Fanuc TP program (LS listing): FM195006.ls

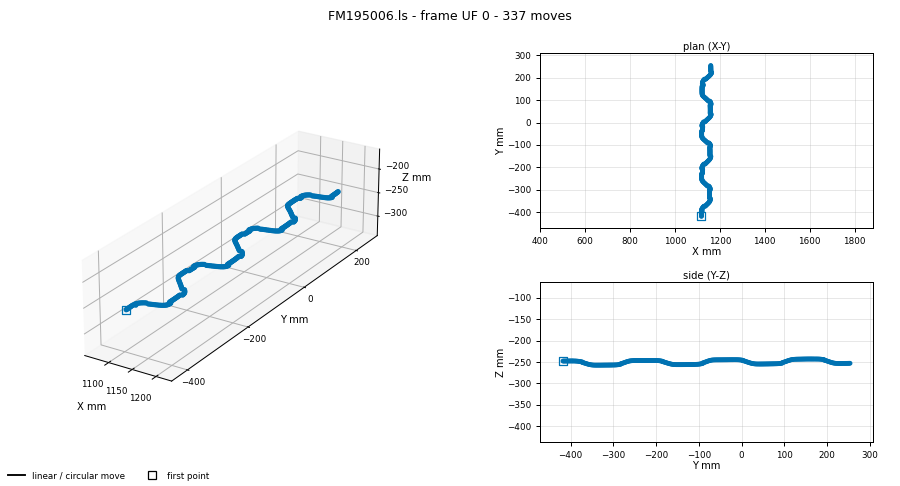
[picture p0: tool path of FM195006.ls in frame UF 0, 337 of 337 moves have a stored position in this frame; points joined in program order, loops and branches not executed]
/PROG  FM195006
/ATTR
OWNER		= MNEDITOR;
COMMENT		= "Auto FANUC move";
PROG_SIZE	= 0;
CREATE		= DATE 26-04-24  TIME 19:50:06;
MODIFIED	= DATE 26-04-24  TIME 19:50:06;
FILE_NAME	= ;
VERSION		= 0;
LINE_COUNT	= 342;
MEMORY_SIZE	= 0;
PROTECT		= READ_WRITE;
TCD:  STACK_SIZE	= 0,
      TASK_PRIORITY	= 50,
      TIME_SLICE	= 0,
      BUSY_LAMP_OFF	= 0,
      ABORT_REQUEST	= 0,
      PAUSE_REQUEST	= 0;
DEFAULT_GROUP	= 1,*,*,*,*;
CONTROL_CODE	= 00000000 00000000;
/MN
   1:  UFRAME_NUM=0 ;
   2:  UTOOL_NUM=1 ;
   3:  R[93]=10 ;
   4:  L P[1] 7mm/sec FINE ;
   5:  L P[2] 7mm/sec FINE ;
   6:  L P[3] 7mm/sec FINE ;
   7:  L P[4] 7mm/sec FINE ;
   8:  L P[5] 7mm/sec FINE ;
   9:  L P[6] 7mm/sec FINE ;
  10:  L P[7] 7mm/sec FINE ;
  11:  L P[8] 7mm/sec FINE ;
  12:  L P[9] 7mm/sec FINE ;
  13:  L P[10] 7mm/sec FINE ;
  14:  L P[11] 7mm/sec FINE ;
  15:  L P[12] 7mm/sec FINE ;
  16:  L P[13] 7mm/sec FINE ;
  17:  L P[14] 7mm/sec FINE ;
  18:  L P[15] 7mm/sec FINE ;
  19:  L P[16] 7mm/sec FINE ;
  20:  L P[17] 7mm/sec FINE ;
  21:  L P[18] 7mm/sec FINE ;
  22:  L P[19] 7mm/sec FINE ;
  23:  L P[20] 7mm/sec FINE ;
  24:  L P[21] 7mm/sec FINE ;
  25:  L P[22] 7mm/sec FINE ;
  26:  L P[23] 7mm/sec FINE ;
  27:  L P[24] 7mm/sec FINE ;
  28:  L P[25] 7mm/sec FINE ;
  29:  L P[26] 7mm/sec FINE ;
  30:  L P[27] 7mm/sec FINE ;
  31:  L P[28] 7mm/sec FINE ;
  32:  L P[29] 7mm/sec FINE ;
  33:  L P[30] 7mm/sec FINE ;
  34:  L P[31] 7mm/sec FINE ;
  35:  L P[32] 7mm/sec FINE ;
  36:  L P[33] 7mm/sec FINE ;
  37:  L P[34] 7mm/sec FINE ;
  38:  L P[35] 7mm/sec FINE ;
  39:  L P[36] 7mm/sec FINE ;
  40:  L P[37] 7mm/sec FINE ;
  41:  L P[38] 7mm/sec FINE ;
  42:  L P[39] 7mm/sec FINE ;
  43:  L P[40] 7mm/sec FINE ;
  44:  L P[41] 7mm/sec FINE ;
  45:  L P[42] 7mm/sec FINE ;
  46:  L P[43] 7mm/sec FINE ;
  47:  L P[44] 7mm/sec FINE ;
  48:  L P[45] 7mm/sec FINE ;
  49:  L P[46] 7mm/sec FINE ;
  50:  L P[47] 7mm/sec FINE ;
  51:  L P[48] 7mm/sec FINE ;
  52:  L P[49] 7mm/sec FINE ;
  53:  L P[50] 7mm/sec FINE ;
  54:  L P[51] 7mm/sec FINE ;
  55:  L P[52] 7mm/sec FINE ;
  56:  L P[53] 7mm/sec FINE ;
  57:  L P[54] 7mm/sec FINE ;
  58:  L P[55] 7mm/sec FINE ;
  59:  L P[56] 7mm/sec FINE ;
  60:  L P[57] 7mm/sec FINE ;
  61:  L P[58] 7mm/sec FINE ;
  62:  L P[59] 7mm/sec FINE ;
  63:  L P[60] 7mm/sec FINE ;
  64:  L P[61] 7mm/sec FINE ;
  65:  L P[62] 7mm/sec FINE ;
  66:  L P[63] 7mm/sec FINE ;
  67:  L P[64] 7mm/sec FINE ;
  68:  L P[65] 7mm/sec FINE ;
  69:  L P[66] 7mm/sec FINE ;
  70:  L P[67] 7mm/sec FINE ;
  71:  L P[68] 7mm/sec FINE ;
  72:  L P[69] 7mm/sec FINE ;
  73:  L P[70] 7mm/sec FINE ;
  74:  L P[71] 7mm/sec FINE ;
  75:  L P[72] 7mm/sec FINE ;
  76:  L P[73] 7mm/sec FINE ;
  77:  L P[74] 7mm/sec FINE ;
  78:  L P[75] 7mm/sec FINE ;
  79:  L P[76] 7mm/sec FINE ;
  80:  L P[77] 7mm/sec FINE ;
  81:  L P[78] 7mm/sec FINE ;
  82:  L P[79] 7mm/sec FINE ;
  83:  L P[80] 7mm/sec FINE ;
  84:  L P[81] 7mm/sec FINE ;
  85:  L P[82] 7mm/sec FINE ;
  86:  L P[83] 7mm/sec FINE ;
  87:  L P[84] 7mm/sec FINE ;
  88:  L P[85] 7mm/sec FINE ;
  89:  L P[86] 7mm/sec FINE ;
  90:  L P[87] 7mm/sec FINE ;
  91:  L P[88] 7mm/sec FINE ;
  92:  L P[89] 7mm/sec FINE ;
  93:  L P[90] 7mm/sec FINE ;
  94:  L P[91] 7mm/sec FINE ;
  95:  L P[92] 7mm/sec FINE ;
  96:  L P[93] 7mm/sec FINE ;
  97:  L P[94] 7mm/sec FINE ;
  98:  L P[95] 7mm/sec FINE ;
  99:  L P[96] 7mm/sec FINE ;
 100:  L P[97] 7mm/sec FINE ;
 101:  L P[98] 7mm/sec FINE ;
 102:  L P[99] 7mm/sec FINE ;
 103:  L P[100] 7mm/sec FINE ;
 104:  L P[101] 7mm/sec FINE ;
 105:  L P[102] 7mm/sec FINE ;
 106:  L P[103] 7mm/sec FINE ;
 107:  L P[104] 7mm/sec FINE ;
 108:  L P[105] 7mm/sec FINE ;
 109:  L P[106] 7mm/sec FINE ;
 110:  L P[107] 7mm/sec FINE ;
 111:  L P[108] 7mm/sec FINE ;
 112:  L P[109] 7mm/sec FINE ;
 113:  L P[110] 7mm/sec FINE ;
 114:  L P[111] 7mm/sec FINE ;
 115:  L P[112] 7mm/sec FINE ;
 116:  L P[113] 7mm/sec FINE ;
 117:  L P[114] 7mm/sec FINE ;
 118:  L P[115] 7mm/sec FINE ;
 119:  L P[116] 7mm/sec FINE ;
 120:  L P[117] 7mm/sec FINE ;
 121:  L P[118] 7mm/sec FINE ;
 122:  L P[119] 7mm/sec FINE ;
 123:  L P[120] 7mm/sec FINE ;
 124:  L P[121] 7mm/sec FINE ;
 125:  L P[122] 7mm/sec FINE ;
 126:  L P[123] 7mm/sec FINE ;
 127:  L P[124] 7mm/sec FINE ;
 128:  L P[125] 7mm/sec FINE ;
 129:  L P[126] 7mm/sec FINE ;
 130:  L P[127] 7mm/sec FINE ;
 131:  L P[128] 7mm/sec FINE ;
 132:  L P[129] 7mm/sec FINE ;
 133:  L P[130] 7mm/sec FINE ;
 134:  L P[131] 7mm/sec FINE ;
 135:  L P[132] 7mm/sec FINE ;
 136:  L P[133] 7mm/sec FINE ;
 137:  L P[134] 7mm/sec FINE ;
 138:  L P[135] 7mm/sec FINE ;
 139:  L P[136] 7mm/sec FINE ;
 140:  L P[137] 7mm/sec FINE ;
 141:  L P[138] 7mm/sec FINE ;
 142:  L P[139] 7mm/sec FINE ;
 143:  L P[140] 7mm/sec FINE ;
 144:  L P[141] 7mm/sec FINE ;
 145:  L P[142] 7mm/sec FINE ;
 146:  L P[143] 7mm/sec FINE ;
 147:  L P[144] 7mm/sec FINE ;
 148:  L P[145] 7mm/sec FINE ;
 149:  L P[146] 7mm/sec FINE ;
 150:  L P[147] 7mm/sec FINE ;
 151:  L P[148] 7mm/sec FINE ;
 152:  L P[149] 7mm/sec FINE ;
 153:  L P[150] 7mm/sec FINE ;
 154:  L P[151] 7mm/sec FINE ;
 155:  L P[152] 7mm/sec FINE ;
 156:  L P[153] 7mm/sec FINE ;
 157:  L P[154] 7mm/sec FINE ;
 158:  L P[155] 7mm/sec FINE ;
 159:  L P[156] 7mm/sec FINE ;
 160:  L P[157] 7mm/sec FINE ;
 161:  L P[158] 7mm/sec FINE ;
 162:  L P[159] 7mm/sec FINE ;
 163:  L P[160] 7mm/sec FINE ;
 164:  L P[161] 7mm/sec FINE ;
 165:  L P[162] 7mm/sec FINE ;
 166:  L P[163] 7mm/sec FINE ;
 167:  L P[164] 7mm/sec FINE ;
 168:  L P[165] 7mm/sec FINE ;
 169:  L P[166] 7mm/sec FINE ;
 170:  L P[167] 7mm/sec FINE ;
 171:  L P[168] 7mm/sec FINE ;
 172:  L P[169] 7mm/sec FINE ;
 173:  L P[170] 7mm/sec FINE ;
 174:  L P[171] 7mm/sec FINE ;
 175:  L P[172] 7mm/sec FINE ;
 176:  L P[173] 7mm/sec FINE ;
 177:  L P[174] 7mm/sec FINE ;
 178:  L P[175] 7mm/sec FINE ;
 179:  L P[176] 7mm/sec FINE ;
 180:  L P[177] 7mm/sec FINE ;
 181:  L P[178] 7mm/sec FINE ;
 182:  L P[179] 7mm/sec FINE ;
 183:  L P[180] 7mm/sec FINE ;
 184:  L P[181] 7mm/sec FINE ;
 185:  L P[182] 7mm/sec FINE ;
 186:  L P[183] 7mm/sec FINE ;
 187:  L P[184] 7mm/sec FINE ;
 188:  L P[185] 7mm/sec FINE ;
 189:  L P[186] 7mm/sec FINE ;
 190:  L P[187] 7mm/sec FINE ;
 191:  L P[188] 7mm/sec FINE ;
 192:  L P[189] 7mm/sec FINE ;
 193:  L P[190] 7mm/sec FINE ;
 194:  L P[191] 7mm/sec FINE ;
 195:  L P[192] 7mm/sec FINE ;
 196:  L P[193] 7mm/sec FINE ;
 197:  L P[194] 7mm/sec FINE ;
 198:  L P[195] 7mm/sec FINE ;
 199:  L P[196] 7mm/sec FINE ;
 200:  L P[197] 7mm/sec FINE ;
 201:  L P[198] 7mm/sec FINE ;
 202:  L P[199] 7mm/sec FINE ;
 203:  L P[200] 7mm/sec FINE ;
 204:  L P[201] 7mm/sec FINE ;
 205:  L P[202] 7mm/sec FINE ;
 206:  L P[203] 7mm/sec FINE ;
 207:  L P[204] 7mm/sec FINE ;
 208:  L P[205] 7mm/sec FINE ;
 209:  L P[206] 7mm/sec FINE ;
 210:  L P[207] 7mm/sec FINE ;
 211:  L P[208] 7mm/sec FINE ;
 212:  L P[209] 7mm/sec FINE ;
 213:  L P[210] 7mm/sec FINE ;
 214:  L P[211] 7mm/sec FINE ;
 215:  L P[212] 7mm/sec FINE ;
 216:  L P[213] 7mm/sec FINE ;
 217:  L P[214] 7mm/sec FINE ;
 218:  L P[215] 7mm/sec FINE ;
 219:  L P[216] 7mm/sec FINE ;
 220:  L P[217] 7mm/sec FINE ;
 221:  L P[218] 7mm/sec FINE ;
 222:  L P[219] 7mm/sec FINE ;
 223:  L P[220] 7mm/sec FINE ;
 224:  L P[221] 7mm/sec FINE ;
 225:  L P[222] 7mm/sec FINE ;
 226:  L P[223] 7mm/sec FINE ;
 227:  L P[224] 7mm/sec FINE ;
 228:  L P[225] 7mm/sec FINE ;
 229:  L P[226] 7mm/sec FINE ;
 230:  L P[227] 7mm/sec FINE ;
 231:  L P[228] 7mm/sec FINE ;
 232:  L P[229] 7mm/sec FINE ;
 233:  L P[230] 7mm/sec FINE ;
 234:  L P[231] 7mm/sec FINE ;
 235:  L P[232] 7mm/sec FINE ;
 236:  L P[233] 7mm/sec FINE ;
 237:  L P[234] 7mm/sec FINE ;
 238:  L P[235] 7mm/sec FINE ;
 239:  L P[236] 7mm/sec FINE ;
 240:  L P[237] 7mm/sec FINE ;
 241:  L P[238] 7mm/sec FINE ;
 242:  L P[239] 7mm/sec FINE ;
 243:  L P[240] 7mm/sec FINE ;
 244:  L P[241] 7mm/sec FINE ;
 245:  L P[242] 7mm/sec FINE ;
 246:  L P[243] 7mm/sec FINE ;
 247:  L P[244] 7mm/sec FINE ;
 248:  L P[245] 7mm/sec FINE ;
 249:  L P[246] 7mm/sec FINE ;
 250:  L P[247] 7mm/sec FINE ;
 251:  L P[248] 7mm/sec FINE ;
 252:  L P[249] 7mm/sec FINE ;
 253:  L P[250] 7mm/sec FINE ;
 254:  L P[251] 7mm/sec FINE ;
 255:  L P[252] 7mm/sec FINE ;
 256:  L P[253] 7mm/sec FINE ;
 257:  L P[254] 7mm/sec FINE ;
 258:  L P[255] 7mm/sec FINE ;
 259:  L P[256] 7mm/sec FINE ;
 260:  L P[257] 7mm/sec FINE ;
 261:  L P[258] 7mm/sec FINE ;
 262:  L P[259] 7mm/sec FINE ;
 263:  L P[260] 7mm/sec FINE ;
 264:  L P[261] 7mm/sec FINE ;
 265:  L P[262] 7mm/sec FINE ;
 266:  L P[263] 7mm/sec FINE ;
 267:  L P[264] 7mm/sec FINE ;
 268:  L P[265] 7mm/sec FINE ;
 269:  L P[266] 7mm/sec FINE ;
 270:  L P[267] 7mm/sec FINE ;
 271:  L P[268] 7mm/sec FINE ;
 272:  L P[269] 7mm/sec FINE ;
 273:  L P[270] 7mm/sec FINE ;
 274:  L P[271] 7mm/sec FINE ;
 275:  L P[272] 7mm/sec FINE ;
 276:  L P[273] 7mm/sec FINE ;
 277:  L P[274] 7mm/sec FINE ;
 278:  L P[275] 7mm/sec FINE ;
 279:  L P[276] 7mm/sec FINE ;
 280:  L P[277] 7mm/sec FINE ;
 281:  L P[278] 7mm/sec FINE ;
 282:  L P[279] 7mm/sec FINE ;
 283:  L P[280] 7mm/sec FINE ;
 284:  L P[281] 7mm/sec FINE ;
 285:  L P[282] 7mm/sec FINE ;
 286:  L P[283] 7mm/sec FINE ;
 287:  L P[284] 7mm/sec FINE ;
 288:  L P[285] 7mm/sec FINE ;
 289:  L P[286] 7mm/sec FINE ;
 290:  L P[287] 7mm/sec FINE ;
 291:  L P[288] 7mm/sec FINE ;
 292:  L P[289] 7mm/sec FINE ;
 293:  L P[290] 7mm/sec FINE ;
 294:  L P[291] 7mm/sec FINE ;
 295:  L P[292] 7mm/sec FINE ;
 296:  L P[293] 7mm/sec FINE ;
 297:  L P[294] 7mm/sec FINE ;
 298:  L P[295] 7mm/sec FINE ;
 299:  L P[296] 7mm/sec FINE ;
 300:  L P[297] 7mm/sec FINE ;
 301:  L P[298] 7mm/sec FINE ;
 302:  L P[299] 7mm/sec FINE ;
 303:  L P[300] 7mm/sec FINE ;
 304:  L P[301] 7mm/sec FINE ;
 305:  L P[302] 7mm/sec FINE ;
 306:  L P[303] 7mm/sec FINE ;
 307:  L P[304] 7mm/sec FINE ;
 308:  L P[305] 7mm/sec FINE ;
 309:  L P[306] 7mm/sec FINE ;
 310:  L P[307] 7mm/sec FINE ;
 311:  L P[308] 7mm/sec FINE ;
 312:  L P[309] 7mm/sec FINE ;
 313:  L P[310] 7mm/sec FINE ;
 314:  L P[311] 7mm/sec FINE ;
 315:  L P[312] 7mm/sec FINE ;
 316:  L P[313] 7mm/sec FINE ;
 317:  L P[314] 7mm/sec FINE ;
 318:  L P[315] 7mm/sec FINE ;
 319:  L P[316] 7mm/sec FINE ;
 320:  L P[317] 7mm/sec FINE ;
 321:  L P[318] 7mm/sec FINE ;
 322:  L P[319] 7mm/sec FINE ;
 323:  L P[320] 7mm/sec FINE ;
 324:  L P[321] 7mm/sec FINE ;
 325:  L P[322] 7mm/sec FINE ;
 326:  L P[323] 7mm/sec FINE ;
 327:  L P[324] 7mm/sec FINE ;
 328:  L P[325] 7mm/sec FINE ;
 329:  L P[326] 7mm/sec FINE ;
 330:  L P[327] 7mm/sec FINE ;
 331:  L P[328] 7mm/sec FINE ;
 332:  L P[329] 7mm/sec FINE ;
 333:  L P[330] 7mm/sec FINE ;
 334:  L P[331] 7mm/sec FINE ;
 335:  L P[332] 7mm/sec FINE ;
 336:  L P[333] 7mm/sec FINE ;
 337:  L P[334] 7mm/sec FINE ;
 338:  L P[335] 7mm/sec FINE ;
 339:  L P[336] 7mm/sec FINE ;
 340:  L P[337] 7mm/sec FINE ;
 341:  R[93]=1 ;
 342:  END ;
/POS
P[1]{
   GP1:
	UF : 0, UT : 1,		CONFIG : 'N U T, 0, 0, 0',
	X = 1117.999  mm,	Y = -418.067  mm,	Z = -247.754  mm,
	W = 0.000 deg,	P = 30.000 deg,	R = 175.494 deg
};
P[2]{
   GP1:
	UF : 0, UT : 1,		CONFIG : 'N U T, 0, 0, 0',
	X = 1117.932  mm,	Y = -416.071  mm,	Z = -247.733  mm,
	W = 0.000 deg,	P = 30.000 deg,	R = 175.494 deg
};
P[3]{
   GP1:
	UF : 0, UT : 1,		CONFIG : 'N U T, 0, 0, 0',
	X = 1117.857  mm,	Y = -414.076  mm,	Z = -247.707  mm,
	W = 0.000 deg,	P = 30.000 deg,	R = 175.494 deg
};
P[4]{
   GP1:
	UF : 0, UT : 1,		CONFIG : 'N U T, 0, 0, 0',
	X = 1117.780  mm,	Y = -412.071  mm,	Z = -247.675  mm,
	W = 0.000 deg,	P = 30.000 deg,	R = 175.494 deg
};
P[5]{
   GP1:
	UF : 0, UT : 1,		CONFIG : 'N U T, 0, 0, 0',
	X = 1117.714  mm,	Y = -410.060  mm,	Z = -247.642  mm,
	W = 0.000 deg,	P = 30.000 deg,	R = 175.494 deg
};
P[6]{
   GP1:
	UF : 0, UT : 1,		CONFIG : 'N U T, 0, 0, 0',
	X = 1117.659  mm,	Y = -408.049  mm,	Z = -247.610  mm,
	W = 0.000 deg,	P = 30.000 deg,	R = 175.494 deg
};
P[7]{
   GP1:
	UF : 0, UT : 1,		CONFIG : 'N U T, 0, 0, 0',
	X = 1117.615  mm,	Y = -406.039  mm,	Z = -247.582  mm,
	W = 0.000 deg,	P = 30.000 deg,	R = 175.494 deg
};
P[8]{
   GP1:
	UF : 0, UT : 1,		CONFIG : 'N U T, 0, 0, 0',
	X = 1117.582  mm,	Y = -404.022  mm,	Z = -247.555  mm,
	W = 0.000 deg,	P = 30.000 deg,	R = 175.494 deg
};
P[9]{
   GP1:
	UF : 0, UT : 1,		CONFIG : 'N U T, 0, 0, 0',
	X = 1117.571  mm,	Y = -402.004  mm,	Z = -247.531  mm,
	W = 0.000 deg,	P = 30.000 deg,	R = 175.494 deg
};
P[10]{
   GP1:
	UF : 0, UT : 1,		CONFIG : 'N U T, 0, 0, 0',
	X = 1117.574  mm,	Y = -399.980  mm,	Z = -247.513  mm,
	W = 0.000 deg,	P = 30.000 deg,	R = 175.494 deg
};
P[11]{
   GP1:
	UF : 0, UT : 1,		CONFIG : 'N U T, 0, 0, 0',
	X = 1117.612  mm,	Y = -397.943  mm,	Z = -247.507  mm,
	W = 0.000 deg,	P = 30.000 deg,	R = 175.494 deg
};
P[12]{
   GP1:
	UF : 0, UT : 1,		CONFIG : 'N U T, 0, 0, 0',
	X = 1117.692  mm,	Y = -395.874  mm,	Z = -247.515  mm,
	W = 0.000 deg,	P = 30.000 deg,	R = 175.494 deg
};
P[13]{
   GP1:
	UF : 0, UT : 1,		CONFIG : 'N U T, 0, 0, 0',
	X = 1121.852  mm,	Y = -394.217  mm,	Z = -247.538  mm,
	W = 0.000 deg,	P = 30.000 deg,	R = 175.494 deg
};
P[14]{
   GP1:
	UF : 0, UT : 1,		CONFIG : 'N U T, 0, 0, 0',
	X = 1118.152  mm,	Y = -391.671  mm,	Z = -247.590  mm,
	W = 0.000 deg,	P = 30.000 deg,	R = 170.031 deg
};
P[15]{
   GP1:
	UF : 0, UT : 1,		CONFIG : 'N U T, 0, 0, 0',
	X = 1118.595  mm,	Y = -389.498  mm,	Z = -247.675  mm,
	W = 0.000 deg,	P = 30.000 deg,	R = 162.233 deg
};
P[16]{
   GP1:
	UF : 0, UT : 1,		CONFIG : 'N U T, 0, 0, 0',
	X = 1119.280  mm,	Y = -387.326  mm,	Z = -247.802  mm,
	W = 0.000 deg,	P = 30.000 deg,	R = 154.209 deg
};
P[17]{
   GP1:
	UF : 0, UT : 1,		CONFIG : 'N U T, 0, 0, 0',
	X = 1120.146  mm,	Y = -385.162  mm,	Z = -247.954  mm,
	W = 0.000 deg,	P = 30.000 deg,	R = 145.966 deg
};
P[18]{
   GP1:
	UF : 0, UT : 1,		CONFIG : 'N U T, 0, 0, 0',
	X = 1121.277  mm,	Y = -383.000  mm,	Z = -248.156  mm,
	W = 0.000 deg,	P = 30.000 deg,	R = 137.314 deg
};
P[19]{
   GP1:
	UF : 0, UT : 1,		CONFIG : 'N U T, 0, 0, 0',
	X = 1122.601  mm,	Y = -380.901  mm,	Z = -248.418  mm,
	W = 0.000 deg,	P = 30.000 deg,	R = 137.314 deg
};
P[20]{
   GP1:
	UF : 0, UT : 1,		CONFIG : 'N U T, 0, 0, 0',
	X = 1124.026  mm,	Y = -378.816  mm,	Z = -248.729  mm,
	W = 0.000 deg,	P = 30.000 deg,	R = 137.314 deg
};
P[21]{
   GP1:
	UF : 0, UT : 1,		CONFIG : 'N U T, 0, 0, 0',
	X = 1125.669  mm,	Y = -376.727  mm,	Z = -249.118  mm,
	W = 0.000 deg,	P = 30.000 deg,	R = 137.314 deg
};
P[22]{
   GP1:
	UF : 0, UT : 1,		CONFIG : 'N U T, 0, 0, 0',
	X = 1127.425  mm,	Y = -374.692  mm,	Z = -249.568  mm,
	W = 0.000 deg,	P = 30.000 deg,	R = 137.314 deg
};
P[23]{
   GP1:
	UF : 0, UT : 1,		CONFIG : 'N U T, 0, 0, 0',
	X = 1129.189  mm,	Y = -372.655  mm,	Z = -250.051  mm,
	W = 0.000 deg,	P = 30.000 deg,	R = 137.314 deg
};
P[24]{
   GP1:
	UF : 0, UT : 1,		CONFIG : 'N U T, 0, 0, 0',
	X = 1134.014  mm,	Y = -373.387  mm,	Z = -250.615  mm,
	W = 0.000 deg,	P = 30.000 deg,	R = 137.314 deg
};
P[25]{
   GP1:
	UF : 0, UT : 1,		CONFIG : 'N U T, 0, 0, 0',
	X = 1135.950  mm,	Y = -371.401  mm,	Z = -251.227  mm,
	W = 0.000 deg,	P = 30.000 deg,	R = 137.314 deg
};
P[26]{
   GP1:
	UF : 0, UT : 1,		CONFIG : 'N U T, 0, 0, 0',
	X = 1137.893  mm,	Y = -369.434  mm,	Z = -251.859  mm,
	W = 0.000 deg,	P = 30.000 deg,	R = 137.314 deg
};
P[27]{
   GP1:
	UF : 0, UT : 1,		CONFIG : 'N U T, 0, 0, 0',
	X = 1140.018  mm,	Y = -367.445  mm,	Z = -252.527  mm,
	W = 0.000 deg,	P = 30.000 deg,	R = 137.314 deg
};
P[28]{
   GP1:
	UF : 0, UT : 1,		CONFIG : 'N U T, 0, 0, 0',
	X = 1142.083  mm,	Y = -365.426  mm,	Z = -253.157  mm,
	W = 0.000 deg,	P = 30.000 deg,	R = 137.314 deg
};
P[29]{
   GP1:
	UF : 0, UT : 1,		CONFIG : 'N U T, 0, 0, 0',
	X = 1144.092  mm,	Y = -363.439  mm,	Z = -253.772  mm,
	W = 0.000 deg,	P = 30.000 deg,	R = 137.314 deg
};
P[30]{
   GP1:
	UF : 0, UT : 1,		CONFIG : 'N U T, 0, 0, 0',
	X = 1146.210  mm,	Y = -361.441  mm,	Z = -254.406  mm,
	W = 0.000 deg,	P = 30.000 deg,	R = 143.831 deg
};
P[31]{
   GP1:
	UF : 0, UT : 1,		CONFIG : 'N U T, 0, 0, 0',
	X = 1148.286  mm,	Y = -359.401  mm,	Z = -255.004  mm,
	W = 0.000 deg,	P = 30.000 deg,	R = 155.941 deg
};
P[32]{
   GP1:
	UF : 0, UT : 1,		CONFIG : 'N U T, 0, 0, 0',
	X = 1150.228  mm,	Y = -357.348  mm,	Z = -255.551  mm,
	W = 0.000 deg,	P = 30.000 deg,	R = 167.597 deg
};
P[33]{
   GP1:
	UF : 0, UT : 1,		CONFIG : 'N U T, 0, 0, 0',
	X = 1152.071  mm,	Y = -355.248  mm,	Z = -256.048  mm,
	W = 0.000 deg,	P = 30.000 deg,	R = 178.845 deg
};
P[34]{
   GP1:
	UF : 0, UT : 1,		CONFIG : 'N U T, 0, 0, 0',
	X = 1153.605  mm,	Y = -353.112  mm,	Z = -256.446  mm,
	W = 0.000 deg,	P = 30.000 deg,	R = 178.845 deg
};
P[35]{
   GP1:
	UF : 0, UT : 1,		CONFIG : 'N U T, 0, 0, 0',
	X = 1154.932  mm,	Y = -350.971  mm,	Z = -256.780  mm,
	W = 0.000 deg,	P = 30.000 deg,	R = 178.845 deg
};
P[36]{
   GP1:
	UF : 0, UT : 1,		CONFIG : 'N U T, 0, 0, 0',
	X = 1156.016  mm,	Y = -348.756  mm,	Z = -257.035  mm,
	W = 0.000 deg,	P = 30.000 deg,	R = 178.845 deg
};
P[37]{
   GP1:
	UF : 0, UT : 1,		CONFIG : 'N U T, 0, 0, 0',
	X = 1156.751  mm,	Y = -346.509  mm,	Z = -257.195  mm,
	W = 0.000 deg,	P = 30.000 deg,	R = 178.845 deg
};
P[38]{
   GP1:
	UF : 0, UT : 1,		CONFIG : 'N U T, 0, 0, 0',
	X = 1157.193  mm,	Y = -344.312  mm,	Z = -257.285  mm,
	W = 0.000 deg,	P = 30.000 deg,	R = 178.845 deg
};
P[39]{
   GP1:
	UF : 0, UT : 1,		CONFIG : 'N U T, 0, 0, 0',
	X = 1157.443  mm,	Y = -342.157  mm,	Z = -257.325  mm,
	W = 0.000 deg,	P = 30.000 deg,	R = 178.845 deg
};
P[40]{
   GP1:
	UF : 0, UT : 1,		CONFIG : 'N U T, 0, 0, 0',
	X = 1157.532  mm,	Y = -340.068  mm,	Z = -257.329  mm,
	W = 0.000 deg,	P = 30.000 deg,	R = 178.845 deg
};
P[41]{
   GP1:
	UF : 0, UT : 1,		CONFIG : 'N U T, 0, 0, 0',
	X = 1157.585  mm,	Y = -338.048  mm,	Z = -257.329  mm,
	W = 0.000 deg,	P = 30.000 deg,	R = 178.845 deg
};
P[42]{
   GP1:
	UF : 0, UT : 1,		CONFIG : 'N U T, 0, 0, 0',
	X = 1153.629  mm,	Y = -335.963  mm,	Z = -257.326  mm,
	W = 0.000 deg,	P = 30.000 deg,	R = 178.845 deg
};
P[43]{
   GP1:
	UF : 0, UT : 1,		CONFIG : 'N U T, 0, 0, 0',
	X = 1153.660  mm,	Y = -333.972  mm,	Z = -257.321  mm,
	W = 0.000 deg,	P = 30.000 deg,	R = 178.845 deg
};
P[44]{
   GP1:
	UF : 0, UT : 1,		CONFIG : 'N U T, 0, 0, 0',
	X = 1153.684  mm,	Y = -331.978  mm,	Z = -257.311  mm,
	W = 0.000 deg,	P = 30.000 deg,	R = 178.845 deg
};
P[45]{
   GP1:
	UF : 0, UT : 1,		CONFIG : 'N U T, 0, 0, 0',
	X = 1153.703  mm,	Y = -329.986  mm,	Z = -257.295  mm,
	W = 0.000 deg,	P = 30.000 deg,	R = 178.845 deg
};
P[46]{
   GP1:
	UF : 0, UT : 1,		CONFIG : 'N U T, 0, 0, 0',
	X = 1153.712  mm,	Y = -327.993  mm,	Z = -257.277  mm,
	W = 0.000 deg,	P = 30.000 deg,	R = 178.845 deg
};
P[47]{
   GP1:
	UF : 0, UT : 1,		CONFIG : 'N U T, 0, 0, 0',
	X = 1153.716  mm,	Y = -325.996  mm,	Z = -257.255  mm,
	W = 0.000 deg,	P = 30.000 deg,	R = 178.845 deg
};
P[48]{
   GP1:
	UF : 0, UT : 1,		CONFIG : 'N U T, 0, 0, 0',
	X = 1153.719  mm,	Y = -323.998  mm,	Z = -257.232  mm,
	W = 0.000 deg,	P = 30.000 deg,	R = 178.845 deg
};
P[49]{
   GP1:
	UF : 0, UT : 1,		CONFIG : 'N U T, 0, 0, 0',
	X = 1153.721  mm,	Y = -321.999  mm,	Z = -257.210  mm,
	W = 0.000 deg,	P = 30.000 deg,	R = 178.845 deg
};
P[50]{
   GP1:
	UF : 0, UT : 1,		CONFIG : 'N U T, 0, 0, 0',
	X = 1153.721  mm,	Y = -320.005  mm,	Z = -257.188  mm,
	W = 0.000 deg,	P = 30.000 deg,	R = 178.845 deg
};
P[51]{
   GP1:
	UF : 0, UT : 1,		CONFIG : 'N U T, 0, 0, 0',
	X = 1153.710  mm,	Y = -318.013  mm,	Z = -257.169  mm,
	W = 0.000 deg,	P = 30.000 deg,	R = 178.845 deg
};
P[52]{
   GP1:
	UF : 0, UT : 1,		CONFIG : 'N U T, 0, 0, 0',
	X = 1153.695  mm,	Y = -316.020  mm,	Z = -257.154  mm,
	W = 0.000 deg,	P = 30.000 deg,	R = 178.845 deg
};
P[53]{
   GP1:
	UF : 0, UT : 1,		CONFIG : 'N U T, 0, 0, 0',
	X = 1153.671  mm,	Y = -314.026  mm,	Z = -257.140  mm,
	W = 0.000 deg,	P = 30.000 deg,	R = 178.845 deg
};
P[54]{
   GP1:
	UF : 0, UT : 1,		CONFIG : 'N U T, 0, 0, 0',
	X = 1153.644  mm,	Y = -312.033  mm,	Z = -257.124  mm,
	W = 0.000 deg,	P = 30.000 deg,	R = 178.845 deg
};
P[55]{
   GP1:
	UF : 0, UT : 1,		CONFIG : 'N U T, 0, 0, 0',
	X = 1153.605  mm,	Y = -310.048  mm,	Z = -257.107  mm,
	W = 0.000 deg,	P = 30.000 deg,	R = 178.845 deg
};
P[56]{
   GP1:
	UF : 0, UT : 1,		CONFIG : 'N U T, 0, 0, 0',
	X = 1153.548  mm,	Y = -308.060  mm,	Z = -257.086  mm,
	W = 0.000 deg,	P = 30.000 deg,	R = 178.845 deg
};
P[57]{
   GP1:
	UF : 0, UT : 1,		CONFIG : 'N U T, 0, 0, 0',
	X = 1153.485  mm,	Y = -306.064  mm,	Z = -257.062  mm,
	W = 0.000 deg,	P = 30.000 deg,	R = 178.845 deg
};
P[58]{
   GP1:
	UF : 0, UT : 1,		CONFIG : 'N U T, 0, 0, 0',
	X = 1153.421  mm,	Y = -304.072  mm,	Z = -257.034  mm,
	W = 0.000 deg,	P = 30.000 deg,	R = 178.845 deg
};
P[59]{
   GP1:
	UF : 0, UT : 1,		CONFIG : 'N U T, 0, 0, 0',
	X = 1153.342  mm,	Y = -302.082  mm,	Z = -257.003  mm,
	W = 0.000 deg,	P = 30.000 deg,	R = 178.845 deg
};
P[60]{
   GP1:
	UF : 0, UT : 1,		CONFIG : 'N U T, 0, 0, 0',
	X = 1157.251  mm,	Y = -299.879  mm,	Z = -256.967  mm,
	W = 0.000 deg,	P = 30.000 deg,	R = -172.841 deg
};
P[61]{
   GP1:
	UF : 0, UT : 1,		CONFIG : 'N U T, 0, 0, 0',
	X = 1157.091  mm,	Y = -297.823  mm,	Z = -256.913  mm,
	W = 0.000 deg,	P = 30.000 deg,	R = -163.968 deg
};
P[62]{
   GP1:
	UF : 0, UT : 1,		CONFIG : 'N U T, 0, 0, 0',
	X = 1156.883  mm,	Y = -295.745  mm,	Z = -256.846  mm,
	W = 0.000 deg,	P = 30.000 deg,	R = -155.076 deg
};
P[63]{
   GP1:
	UF : 0, UT : 1,		CONFIG : 'N U T, 0, 0, 0',
	X = 1156.543  mm,	Y = -293.588  mm,	Z = -256.745  mm,
	W = 0.000 deg,	P = 30.000 deg,	R = -146.113 deg
};
P[64]{
   GP1:
	UF : 0, UT : 1,		CONFIG : 'N U T, 0, 0, 0',
	X = 1155.946  mm,	Y = -291.342  mm,	Z = -256.580  mm,
	W = 0.000 deg,	P = 30.000 deg,	R = -136.938 deg
};
P[65]{
   GP1:
	UF : 0, UT : 1,		CONFIG : 'N U T, 0, 0, 0',
	X = 1154.950  mm,	Y = -289.046  mm,	Z = -256.318  mm,
	W = 0.000 deg,	P = 30.000 deg,	R = -136.938 deg
};
P[66]{
   GP1:
	UF : 0, UT : 1,		CONFIG : 'N U T, 0, 0, 0',
	X = 1153.530  mm,	Y = -286.860  mm,	Z = -255.916  mm,
	W = 0.000 deg,	P = 30.000 deg,	R = -136.938 deg
};
P[67]{
   GP1:
	UF : 0, UT : 1,		CONFIG : 'N U T, 0, 0, 0',
	X = 1151.985  mm,	Y = -284.759  mm,	Z = -255.467  mm,
	W = 0.000 deg,	P = 30.000 deg,	R = -136.938 deg
};
P[68]{
   GP1:
	UF : 0, UT : 1,		CONFIG : 'N U T, 0, 0, 0',
	X = 1150.225  mm,	Y = -282.682  mm,	Z = -254.945  mm,
	W = 0.000 deg,	P = 30.000 deg,	R = -136.938 deg
};
P[69]{
   GP1:
	UF : 0, UT : 1,		CONFIG : 'N U T, 0, 0, 0',
	X = 1145.453  mm,	Y = -283.369  mm,	Z = -254.386  mm,
	W = 0.000 deg,	P = 30.000 deg,	R = -136.938 deg
};
P[70]{
   GP1:
	UF : 0, UT : 1,		CONFIG : 'N U T, 0, 0, 0',
	X = 1143.577  mm,	Y = -281.438  mm,	Z = -253.781  mm,
	W = 0.000 deg,	P = 30.000 deg,	R = -136.938 deg
};
P[71]{
   GP1:
	UF : 0, UT : 1,		CONFIG : 'N U T, 0, 0, 0',
	X = 1141.392  mm,	Y = -279.447  mm,	Z = -253.092  mm,
	W = 0.000 deg,	P = 30.000 deg,	R = -136.938 deg
};
P[72]{
   GP1:
	UF : 0, UT : 1,		CONFIG : 'N U T, 0, 0, 0',
	X = 1139.366  mm,	Y = -277.421  mm,	Z = -252.452  mm,
	W = 0.000 deg,	P = 30.000 deg,	R = -136.938 deg
};
P[73]{
   GP1:
	UF : 0, UT : 1,		CONFIG : 'N U T, 0, 0, 0',
	X = 1137.351  mm,	Y = -275.446  mm,	Z = -251.780  mm,
	W = 0.000 deg,	P = 30.000 deg,	R = -136.938 deg
};
P[74]{
   GP1:
	UF : 0, UT : 1,		CONFIG : 'N U T, 0, 0, 0',
	X = 1135.216  mm,	Y = -273.455  mm,	Z = -251.043  mm,
	W = 0.000 deg,	P = 30.000 deg,	R = -136.938 deg
};
P[75]{
   GP1:
	UF : 0, UT : 1,		CONFIG : 'N U T, 0, 0, 0',
	X = 1133.147  mm,	Y = -271.482  mm,	Z = -250.323  mm,
	W = 0.000 deg,	P = 30.000 deg,	R = -136.938 deg
};
P[76]{
   GP1:
	UF : 0, UT : 1,		CONFIG : 'N U T, 0, 0, 0',
	X = 1130.846  mm,	Y = -269.496  mm,	Z = -249.596  mm,
	W = 0.000 deg,	P = 30.000 deg,	R = -136.938 deg
};
P[77]{
   GP1:
	UF : 0, UT : 1,		CONFIG : 'N U T, 0, 0, 0',
	X = 1128.600  mm,	Y = -267.443  mm,	Z = -248.935  mm,
	W = 0.000 deg,	P = 30.000 deg,	R = -144.465 deg
};
P[78]{
   GP1:
	UF : 0, UT : 1,		CONFIG : 'N U T, 0, 0, 0',
	X = 1126.581  mm,	Y = -265.403  mm,	Z = -248.356  mm,
	W = 0.000 deg,	P = 30.000 deg,	R = -156.971 deg
};
P[79]{
   GP1:
	UF : 0, UT : 1,		CONFIG : 'N U T, 0, 0, 0',
	X = 1124.538  mm,	Y = -263.312  mm,	Z = -247.787  mm,
	W = 0.000 deg,	P = 30.000 deg,	R = -169.411 deg
};
P[80]{
   GP1:
	UF : 0, UT : 1,		CONFIG : 'N U T, 0, 0, 0',
	X = 1122.883  mm,	Y = -261.136  mm,	Z = -247.389  mm,
	W = 0.000 deg,	P = 30.000 deg,	R = 179.517 deg
};
P[81]{
   GP1:
	UF : 0, UT : 1,		CONFIG : 'N U T, 0, 0, 0',
	X = 1121.541  mm,	Y = -258.975  mm,	Z = -247.111  mm,
	W = 0.000 deg,	P = 30.000 deg,	R = 179.517 deg
};
P[82]{
   GP1:
	UF : 0, UT : 1,		CONFIG : 'N U T, 0, 0, 0',
	X = 1120.437  mm,	Y = -256.742  mm,	Z = -246.905  mm,
	W = 0.000 deg,	P = 30.000 deg,	R = 179.517 deg
};
P[83]{
   GP1:
	UF : 0, UT : 1,		CONFIG : 'N U T, 0, 0, 0',
	X = 1119.757  mm,	Y = -254.518  mm,	Z = -246.756  mm,
	W = 0.000 deg,	P = 30.000 deg,	R = 179.517 deg
};
P[84]{
   GP1:
	UF : 0, UT : 1,		CONFIG : 'N U T, 0, 0, 0',
	X = 1119.249  mm,	Y = -252.332  mm,	Z = -246.621  mm,
	W = 0.000 deg,	P = 30.000 deg,	R = 179.517 deg
};
P[85]{
   GP1:
	UF : 0, UT : 1,		CONFIG : 'N U T, 0, 0, 0',
	X = 1119.021  mm,	Y = -250.140  mm,	Z = -246.556  mm,
	W = 0.000 deg,	P = 30.000 deg,	R = 179.517 deg
};
P[86]{
   GP1:
	UF : 0, UT : 1,		CONFIG : 'N U T, 0, 0, 0',
	X = 1118.942  mm,	Y = -248.044  mm,	Z = -246.528  mm,
	W = 0.000 deg,	P = 30.000 deg,	R = 179.517 deg
};
P[87]{
   GP1:
	UF : 0, UT : 1,		CONFIG : 'N U T, 0, 0, 0',
	X = 1118.928  mm,	Y = -246.009  mm,	Z = -246.504  mm,
	W = 0.000 deg,	P = 30.000 deg,	R = 179.517 deg
};
P[88]{
   GP1:
	UF : 0, UT : 1,		CONFIG : 'N U T, 0, 0, 0',
	X = 1118.924  mm,	Y = -244.003  mm,	Z = -246.479  mm,
	W = 0.000 deg,	P = 30.000 deg,	R = 179.517 deg
};
P[89]{
   GP1:
	UF : 0, UT : 1,		CONFIG : 'N U T, 0, 0, 0',
	X = 1118.923  mm,	Y = -241.999  mm,	Z = -246.458  mm,
	W = 0.000 deg,	P = 30.000 deg,	R = 179.517 deg
};
P[90]{
   GP1:
	UF : 0, UT : 1,		CONFIG : 'N U T, 0, 0, 0',
	X = 1118.925  mm,	Y = -239.998  mm,	Z = -246.441  mm,
	W = 0.000 deg,	P = 30.000 deg,	R = 179.517 deg
};
P[91]{
   GP1:
	UF : 0, UT : 1,		CONFIG : 'N U T, 0, 0, 0',
	X = 1118.927  mm,	Y = -237.997  mm,	Z = -246.426  mm,
	W = 0.000 deg,	P = 30.000 deg,	R = 179.517 deg
};
P[92]{
   GP1:
	UF : 0, UT : 1,		CONFIG : 'N U T, 0, 0, 0',
	X = 1118.930  mm,	Y = -235.996  mm,	Z = -246.406  mm,
	W = 0.000 deg,	P = 30.000 deg,	R = 179.517 deg
};
P[93]{
   GP1:
	UF : 0, UT : 1,		CONFIG : 'N U T, 0, 0, 0',
	X = 1118.935  mm,	Y = -233.995  mm,	Z = -246.388  mm,
	W = 0.000 deg,	P = 30.000 deg,	R = 179.517 deg
};
P[94]{
   GP1:
	UF : 0, UT : 1,		CONFIG : 'N U T, 0, 0, 0',
	X = 1118.941  mm,	Y = -231.994  mm,	Z = -246.372  mm,
	W = 0.000 deg,	P = 30.000 deg,	R = 179.517 deg
};
P[95]{
   GP1:
	UF : 0, UT : 1,		CONFIG : 'N U T, 0, 0, 0',
	X = 1118.947  mm,	Y = -229.993  mm,	Z = -246.357  mm,
	W = 0.000 deg,	P = 30.000 deg,	R = 179.517 deg
};
P[96]{
   GP1:
	UF : 0, UT : 1,		CONFIG : 'N U T, 0, 0, 0',
	X = 1118.955  mm,	Y = -227.988  mm,	Z = -246.340  mm,
	W = 0.000 deg,	P = 30.000 deg,	R = 179.517 deg
};
P[97]{
   GP1:
	UF : 0, UT : 1,		CONFIG : 'N U T, 0, 0, 0',
	X = 1122.972  mm,	Y = -226.021  mm,	Z = -246.323  mm,
	W = 0.000 deg,	P = 30.000 deg,	R = 179.517 deg
};
P[98]{
   GP1:
	UF : 0, UT : 1,		CONFIG : 'N U T, 0, 0, 0',
	X = 1122.997  mm,	Y = -224.029  mm,	Z = -246.302  mm,
	W = 0.000 deg,	P = 30.000 deg,	R = 179.517 deg
};
P[99]{
   GP1:
	UF : 0, UT : 1,		CONFIG : 'N U T, 0, 0, 0',
	X = 1123.029  mm,	Y = -222.034  mm,	Z = -246.287  mm,
	W = 0.000 deg,	P = 30.000 deg,	R = 179.517 deg
};
P[100]{
   GP1:
	UF : 0, UT : 1,		CONFIG : 'N U T, 0, 0, 0',
	X = 1123.065  mm,	Y = -220.043  mm,	Z = -246.273  mm,
	W = 0.000 deg,	P = 30.000 deg,	R = 179.517 deg
};
P[101]{
   GP1:
	UF : 0, UT : 1,		CONFIG : 'N U T, 0, 0, 0',
	X = 1123.116  mm,	Y = -218.053  mm,	Z = -246.260  mm,
	W = 0.000 deg,	P = 30.000 deg,	R = 179.517 deg
};
P[102]{
   GP1:
	UF : 0, UT : 1,		CONFIG : 'N U T, 0, 0, 0',
	X = 1123.170  mm,	Y = -216.059  mm,	Z = -246.250  mm,
	W = 0.000 deg,	P = 30.000 deg,	R = 179.517 deg
};
P[103]{
   GP1:
	UF : 0, UT : 1,		CONFIG : 'N U T, 0, 0, 0',
	X = 1123.234  mm,	Y = -214.068  mm,	Z = -246.243  mm,
	W = 0.000 deg,	P = 30.000 deg,	R = 179.517 deg
};
P[104]{
   GP1:
	UF : 0, UT : 1,		CONFIG : 'N U T, 0, 0, 0',
	X = 1123.304  mm,	Y = -212.079  mm,	Z = -246.241  mm,
	W = 0.000 deg,	P = 30.000 deg,	R = 179.517 deg
};
P[105]{
   GP1:
	UF : 0, UT : 1,		CONFIG : 'N U T, 0, 0, 0',
	X = 1123.390  mm,	Y = -210.099  mm,	Z = -246.248  mm,
	W = 0.000 deg,	P = 30.000 deg,	R = 179.517 deg
};
P[106]{
   GP1:
	UF : 0, UT : 1,		CONFIG : 'N U T, 0, 0, 0',
	X = 1123.499  mm,	Y = -208.130  mm,	Z = -246.261  mm,
	W = 0.000 deg,	P = 30.000 deg,	R = 179.517 deg
};
P[107]{
   GP1:
	UF : 0, UT : 1,		CONFIG : 'N U T, 0, 0, 0',
	X = 1119.659  mm,	Y = -205.835  mm,	Z = -246.287  mm,
	W = 0.000 deg,	P = 30.000 deg,	R = 171.938 deg
};
P[108]{
   GP1:
	UF : 0, UT : 1,		CONFIG : 'N U T, 0, 0, 0',
	X = 1119.847  mm,	Y = -203.782  mm,	Z = -246.318  mm,
	W = 0.000 deg,	P = 30.000 deg,	R = 163.727 deg
};
P[109]{
   GP1:
	UF : 0, UT : 1,		CONFIG : 'N U T, 0, 0, 0',
	X = 1120.114  mm,	Y = -201.694  mm,	Z = -246.368  mm,
	W = 0.000 deg,	P = 30.000 deg,	R = 155.482 deg
};
P[110]{
   GP1:
	UF : 0, UT : 1,		CONFIG : 'N U T, 0, 0, 0',
	X = 1120.509  mm,	Y = -199.539  mm,	Z = -246.440  mm,
	W = 0.000 deg,	P = 30.000 deg,	R = 147.166 deg
};
P[111]{
   GP1:
	UF : 0, UT : 1,		CONFIG : 'N U T, 0, 0, 0',
	X = 1121.143  mm,	Y = -197.359  mm,	Z = -246.558  mm,
	W = 0.000 deg,	P = 30.000 deg,	R = 138.638 deg
};
P[112]{
   GP1:
	UF : 0, UT : 1,		CONFIG : 'N U T, 0, 0, 0',
	X = 1121.983  mm,	Y = -195.184  mm,	Z = -246.722  mm,
	W = 0.000 deg,	P = 30.000 deg,	R = 138.638 deg
};
P[113]{
   GP1:
	UF : 0, UT : 1,		CONFIG : 'N U T, 0, 0, 0',
	X = 1123.085  mm,	Y = -193.015  mm,	Z = -246.925  mm,
	W = 0.000 deg,	P = 30.000 deg,	R = 138.638 deg
};
P[114]{
   GP1:
	UF : 0, UT : 1,		CONFIG : 'N U T, 0, 0, 0',
	X = 1124.394  mm,	Y = -190.912  mm,	Z = -247.186  mm,
	W = 0.000 deg,	P = 30.000 deg,	R = 138.638 deg
};
P[115]{
   GP1:
	UF : 0, UT : 1,		CONFIG : 'N U T, 0, 0, 0',
	X = 1125.807  mm,	Y = -188.818  mm,	Z = -247.496  mm,
	W = 0.000 deg,	P = 30.000 deg,	R = 138.638 deg
};
P[116]{
   GP1:
	UF : 0, UT : 1,		CONFIG : 'N U T, 0, 0, 0',
	X = 1127.467  mm,	Y = -186.716  mm,	Z = -247.890  mm,
	W = 0.000 deg,	P = 30.000 deg,	R = 138.638 deg
};
P[117]{
   GP1:
	UF : 0, UT : 1,		CONFIG : 'N U T, 0, 0, 0',
	X = 1129.261  mm,	Y = -184.686  mm,	Z = -248.372  mm,
	W = 0.000 deg,	P = 30.000 deg,	R = 138.638 deg
};
P[118]{
   GP1:
	UF : 0, UT : 1,		CONFIG : 'N U T, 0, 0, 0',
	X = 1133.983  mm,	Y = -185.329  mm,	Z = -248.858  mm,
	W = 0.000 deg,	P = 30.000 deg,	R = 138.638 deg
};
P[119]{
   GP1:
	UF : 0, UT : 1,		CONFIG : 'N U T, 0, 0, 0',
	X = 1135.782  mm,	Y = -183.372  mm,	Z = -249.400  mm,
	W = 0.000 deg,	P = 30.000 deg,	R = 138.638 deg
};
P[120]{
   GP1:
	UF : 0, UT : 1,		CONFIG : 'N U T, 0, 0, 0',
	X = 1137.694  mm,	Y = -181.394  mm,	Z = -250.004  mm,
	W = 0.000 deg,	P = 30.000 deg,	R = 138.638 deg
};
P[121]{
   GP1:
	UF : 0, UT : 1,		CONFIG : 'N U T, 0, 0, 0',
	X = 1139.617  mm,	Y = -179.424  mm,	Z = -250.628  mm,
	W = 0.000 deg,	P = 30.000 deg,	R = 138.638 deg
};
P[122]{
   GP1:
	UF : 0, UT : 1,		CONFIG : 'N U T, 0, 0, 0',
	X = 1141.713  mm,	Y = -177.429  mm,	Z = -251.290  mm,
	W = 0.000 deg,	P = 30.000 deg,	R = 138.638 deg
};
P[123]{
   GP1:
	UF : 0, UT : 1,		CONFIG : 'N U T, 0, 0, 0',
	X = 1143.721  mm,	Y = -175.406  mm,	Z = -251.904  mm,
	W = 0.000 deg,	P = 30.000 deg,	R = 138.638 deg
};
P[124]{
   GP1:
	UF : 0, UT : 1,		CONFIG : 'N U T, 0, 0, 0',
	X = 1145.674  mm,	Y = -173.425  mm,	Z = -252.487  mm,
	W = 0.000 deg,	P = 30.000 deg,	R = 144.085 deg
};
P[125]{
   GP1:
	UF : 0, UT : 1,		CONFIG : 'N U T, 0, 0, 0',
	X = 1147.766  mm,	Y = -171.426  mm,	Z = -253.102  mm,
	W = 0.000 deg,	P = 30.000 deg,	R = 155.718 deg
};
P[126]{
   GP1:
	UF : 0, UT : 1,		CONFIG : 'N U T, 0, 0, 0',
	X = 1149.782  mm,	Y = -169.385  mm,	Z = -253.677  mm,
	W = 0.000 deg,	P = 30.000 deg,	R = 166.997 deg
};
P[127]{
   GP1:
	UF : 0, UT : 1,		CONFIG : 'N U T, 0, 0, 0',
	X = 1151.679  mm,	Y = -167.347  mm,	Z = -254.219  mm,
	W = 0.000 deg,	P = 30.000 deg,	R = 177.947 deg
};
P[128]{
   GP1:
	UF : 0, UT : 1,		CONFIG : 'N U T, 0, 0, 0',
	X = 1153.526  mm,	Y = -165.273  mm,	Z = -254.722  mm,
	W = 0.000 deg,	P = 30.000 deg,	R = 177.947 deg
};
P[129]{
   GP1:
	UF : 0, UT : 1,		CONFIG : 'N U T, 0, 0, 0',
	X = 1155.126  mm,	Y = -163.165  mm,	Z = -255.141  mm,
	W = 0.000 deg,	P = 30.000 deg,	R = 177.947 deg
};
P[130]{
   GP1:
	UF : 0, UT : 1,		CONFIG : 'N U T, 0, 0, 0',
	X = 1156.560  mm,	Y = -161.036  mm,	Z = -255.504  mm,
	W = 0.000 deg,	P = 30.000 deg,	R = 177.947 deg
};
P[131]{
   GP1:
	UF : 0, UT : 1,		CONFIG : 'N U T, 0, 0, 0',
	X = 1157.737  mm,	Y = -158.843  mm,	Z = -255.790  mm,
	W = 0.000 deg,	P = 30.000 deg,	R = 177.947 deg
};
P[132]{
   GP1:
	UF : 0, UT : 1,		CONFIG : 'N U T, 0, 0, 0',
	X = 1158.603  mm,	Y = -156.644  mm,	Z = -255.988  mm,
	W = 0.000 deg,	P = 30.000 deg,	R = 177.947 deg
};
P[133]{
   GP1:
	UF : 0, UT : 1,		CONFIG : 'N U T, 0, 0, 0',
	X = 1159.236  mm,	Y = -154.439  mm,	Z = -256.122  mm,
	W = 0.000 deg,	P = 30.000 deg,	R = 177.947 deg
};
P[134]{
   GP1:
	UF : 0, UT : 1,		CONFIG : 'N U T, 0, 0, 0',
	X = 1159.598  mm,	Y = -152.220  mm,	Z = -256.185  mm,
	W = 0.000 deg,	P = 30.000 deg,	R = 177.947 deg
};
P[135]{
   GP1:
	UF : 0, UT : 1,		CONFIG : 'N U T, 0, 0, 0',
	X = 1159.726  mm,	Y = -150.098  mm,	Z = -256.194  mm,
	W = 0.000 deg,	P = 30.000 deg,	R = 177.947 deg
};
P[136]{
   GP1:
	UF : 0, UT : 1,		CONFIG : 'N U T, 0, 0, 0',
	X = 1155.808  mm,	Y = -147.932  mm,	Z = -256.196  mm,
	W = 0.000 deg,	P = 30.000 deg,	R = 177.947 deg
};
P[137]{
   GP1:
	UF : 0, UT : 1,		CONFIG : 'N U T, 0, 0, 0',
	X = 1155.865  mm,	Y = -145.953  mm,	Z = -256.197  mm,
	W = 0.000 deg,	P = 30.000 deg,	R = 177.947 deg
};
P[138]{
   GP1:
	UF : 0, UT : 1,		CONFIG : 'N U T, 0, 0, 0',
	X = 1155.901  mm,	Y = -143.972  mm,	Z = -256.195  mm,
	W = 0.000 deg,	P = 30.000 deg,	R = 177.947 deg
};
P[139]{
   GP1:
	UF : 0, UT : 1,		CONFIG : 'N U T, 0, 0, 0',
	X = 1155.921  mm,	Y = -141.982  mm,	Z = -256.191  mm,
	W = 0.000 deg,	P = 30.000 deg,	R = 177.947 deg
};
P[140]{
   GP1:
	UF : 0, UT : 1,		CONFIG : 'N U T, 0, 0, 0',
	X = 1155.937  mm,	Y = -139.989  mm,	Z = -256.184  mm,
	W = 0.000 deg,	P = 30.000 deg,	R = 177.947 deg
};
P[141]{
   GP1:
	UF : 0, UT : 1,		CONFIG : 'N U T, 0, 0, 0',
	X = 1155.944  mm,	Y = -137.997  mm,	Z = -256.176  mm,
	W = 0.000 deg,	P = 30.000 deg,	R = 177.947 deg
};
P[142]{
   GP1:
	UF : 0, UT : 1,		CONFIG : 'N U T, 0, 0, 0',
	X = 1155.944  mm,	Y = -136.000  mm,	Z = -256.157  mm,
	W = 0.000 deg,	P = 30.000 deg,	R = 177.947 deg
};
P[143]{
   GP1:
	UF : 0, UT : 1,		CONFIG : 'N U T, 0, 0, 0',
	X = 1155.943  mm,	Y = -134.001  mm,	Z = -256.133  mm,
	W = 0.000 deg,	P = 30.000 deg,	R = 177.947 deg
};
P[144]{
   GP1:
	UF : 0, UT : 1,		CONFIG : 'N U T, 0, 0, 0',
	X = 1155.942  mm,	Y = -132.002  mm,	Z = -256.103  mm,
	W = 0.000 deg,	P = 30.000 deg,	R = 177.947 deg
};
P[145]{
   GP1:
	UF : 0, UT : 1,		CONFIG : 'N U T, 0, 0, 0',
	X = 1155.940  mm,	Y = -130.005  mm,	Z = -256.068  mm,
	W = 0.000 deg,	P = 30.000 deg,	R = 177.947 deg
};
P[146]{
   GP1:
	UF : 0, UT : 1,		CONFIG : 'N U T, 0, 0, 0',
	X = 1155.932  mm,	Y = -128.012  mm,	Z = -256.029  mm,
	W = 0.000 deg,	P = 30.000 deg,	R = 177.947 deg
};
P[147]{
   GP1:
	UF : 0, UT : 1,		CONFIG : 'N U T, 0, 0, 0',
	X = 1155.916  mm,	Y = -126.022  mm,	Z = -255.991  mm,
	W = 0.000 deg,	P = 30.000 deg,	R = 177.947 deg
};
P[148]{
   GP1:
	UF : 0, UT : 1,		CONFIG : 'N U T, 0, 0, 0',
	X = 1155.889  mm,	Y = -124.032  mm,	Z = -255.948  mm,
	W = 0.000 deg,	P = 30.000 deg,	R = 177.947 deg
};
P[149]{
   GP1:
	UF : 0, UT : 1,		CONFIG : 'N U T, 0, 0, 0',
	X = 1155.853  mm,	Y = -122.044  mm,	Z = -255.909  mm,
	W = 0.000 deg,	P = 30.000 deg,	R = 177.947 deg
};
P[150]{
   GP1:
	UF : 0, UT : 1,		CONFIG : 'N U T, 0, 0, 0',
	X = 1155.802  mm,	Y = -120.056  mm,	Z = -255.865  mm,
	W = 0.000 deg,	P = 30.000 deg,	R = 177.947 deg
};
P[151]{
   GP1:
	UF : 0, UT : 1,		CONFIG : 'N U T, 0, 0, 0',
	X = 1155.743  mm,	Y = -118.073  mm,	Z = -255.825  mm,
	W = 0.000 deg,	P = 30.000 deg,	R = 177.947 deg
};
P[152]{
   GP1:
	UF : 0, UT : 1,		CONFIG : 'N U T, 0, 0, 0',
	X = 1155.658  mm,	Y = -116.103  mm,	Z = -255.780  mm,
	W = 0.000 deg,	P = 30.000 deg,	R = 177.947 deg
};
P[153]{
   GP1:
	UF : 0, UT : 1,		CONFIG : 'N U T, 0, 0, 0',
	X = 1155.540  mm,	Y = -114.132  mm,	Z = -255.730  mm,
	W = 0.000 deg,	P = 30.000 deg,	R = 177.947 deg
};
P[154]{
   GP1:
	UF : 0, UT : 1,		CONFIG : 'N U T, 0, 0, 0',
	X = 1155.397  mm,	Y = -112.149  mm,	Z = -255.665  mm,
	W = 0.000 deg,	P = 30.000 deg,	R = 177.947 deg
};
P[155]{
   GP1:
	UF : 0, UT : 1,		CONFIG : 'N U T, 0, 0, 0',
	X = 1155.244  mm,	Y = -110.172  mm,	Z = -255.600  mm,
	W = 0.000 deg,	P = 30.000 deg,	R = 177.947 deg
};
P[156]{
   GP1:
	UF : 0, UT : 1,		CONFIG : 'N U T, 0, 0, 0',
	X = 1155.060  mm,	Y = -108.239  mm,	Z = -255.526  mm,
	W = 0.000 deg,	P = 30.000 deg,	R = -173.611 deg
};
P[157]{
   GP1:
	UF : 0, UT : 1,		CONFIG : 'N U T, 0, 0, 0',
	X = 1158.729  mm,	Y = -105.672  mm,	Z = -255.420  mm,
	W = 0.000 deg,	P = 30.000 deg,	R = -163.999 deg
};
P[158]{
   GP1:
	UF : 0, UT : 1,		CONFIG : 'N U T, 0, 0, 0',
	X = 1158.347  mm,	Y = -103.630  mm,	Z = -255.288  mm,
	W = 0.000 deg,	P = 30.000 deg,	R = -154.313 deg
};
P[159]{
   GP1:
	UF : 0, UT : 1,		CONFIG : 'N U T, 0, 0, 0',
	X = 1157.939  mm,	Y = -101.494  mm,	Z = -255.159  mm,
	W = 0.000 deg,	P = 30.000 deg,	R = -144.626 deg
};
P[160]{
   GP1:
	UF : 0, UT : 1,		CONFIG : 'N U T, 0, 0, 0',
	X = 1157.183  mm,	Y = -99.236  mm,	Z = -254.937  mm,
	W = 0.000 deg,	P = 30.000 deg,	R = -134.552 deg
};
P[161]{
   GP1:
	UF : 0, UT : 1,		CONFIG : 'N U T, 0, 0, 0',
	X = 1156.107  mm,	Y = -97.046  mm,	Z = -254.626  mm,
	W = 0.000 deg,	P = 30.000 deg,	R = -134.552 deg
};
P[162]{
   GP1:
	UF : 0, UT : 1,		CONFIG : 'N U T, 0, 0, 0',
	X = 1154.769  mm,	Y = -94.809  mm,	Z = -254.255  mm,
	W = 0.000 deg,	P = 30.000 deg,	R = -134.552 deg
};
P[163]{
   GP1:
	UF : 0, UT : 1,		CONFIG : 'N U T, 0, 0, 0',
	X = 1152.885  mm,	Y = -92.678  mm,	Z = -253.691  mm,
	W = 0.000 deg,	P = 30.000 deg,	R = -134.552 deg
};
P[164]{
   GP1:
	UF : 0, UT : 1,		CONFIG : 'N U T, 0, 0, 0',
	X = 1151.072  mm,	Y = -90.603  mm,	Z = -253.141  mm,
	W = 0.000 deg,	P = 30.000 deg,	R = -134.552 deg
};
P[165]{
   GP1:
	UF : 0, UT : 1,		CONFIG : 'N U T, 0, 0, 0',
	X = 1146.122  mm,	Y = -91.471  mm,	Z = -252.452  mm,
	W = 0.000 deg,	P = 30.000 deg,	R = -134.552 deg
};
P[166]{
   GP1:
	UF : 0, UT : 1,		CONFIG : 'N U T, 0, 0, 0',
	X = 1143.930  mm,	Y = -89.456  mm,	Z = -251.757  mm,
	W = 0.000 deg,	P = 30.000 deg,	R = -134.552 deg
};
P[167]{
   GP1:
	UF : 0, UT : 1,		CONFIG : 'N U T, 0, 0, 0',
	X = 1141.885  mm,	Y = -87.481  mm,	Z = -251.097  mm,
	W = 0.000 deg,	P = 30.000 deg,	R = -134.552 deg
};
P[168]{
   GP1:
	UF : 0, UT : 1,		CONFIG : 'N U T, 0, 0, 0',
	X = 1139.564  mm,	Y = -85.492  mm,	Z = -250.325  mm,
	W = 0.000 deg,	P = 30.000 deg,	R = -134.552 deg
};
P[169]{
   GP1:
	UF : 0, UT : 1,		CONFIG : 'N U T, 0, 0, 0',
	X = 1137.366  mm,	Y = -83.447  mm,	Z = -249.605  mm,
	W = 0.000 deg,	P = 30.000 deg,	R = -134.552 deg
};
P[170]{
   GP1:
	UF : 0, UT : 1,		CONFIG : 'N U T, 0, 0, 0',
	X = 1135.396  mm,	Y = -81.511  mm,	Z = -248.899  mm,
	W = 0.000 deg,	P = 30.000 deg,	R = -134.552 deg
};
P[171]{
   GP1:
	UF : 0, UT : 1,		CONFIG : 'N U T, 0, 0, 0',
	X = 1132.837  mm,	Y = -79.526  mm,	Z = -248.121  mm,
	W = 0.000 deg,	P = 30.000 deg,	R = -134.552 deg
};
P[172]{
   GP1:
	UF : 0, UT : 1,		CONFIG : 'N U T, 0, 0, 0',
	X = 1130.664  mm,	Y = -77.500  mm,	Z = -247.484  mm,
	W = 0.000 deg,	P = 30.000 deg,	R = -139.413 deg
};
P[173]{
   GP1:
	UF : 0, UT : 1,		CONFIG : 'N U T, 0, 0, 0',
	X = 1128.289  mm,	Y = -75.514  mm,	Z = -246.805  mm,
	W = 0.000 deg,	P = 30.000 deg,	R = -154.113 deg
};
P[174]{
   GP1:
	UF : 0, UT : 1,		CONFIG : 'N U T, 0, 0, 0',
	X = 1125.937  mm,	Y = -73.412  mm,	Z = -246.188  mm,
	W = 0.000 deg,	P = 30.000 deg,	R = -168.249 deg
};
P[175]{
   GP1:
	UF : 0, UT : 1,		CONFIG : 'N U T, 0, 0, 0',
	X = 1124.097  mm,	Y = -71.312  mm,	Z = -245.775  mm,
	W = 0.000 deg,	P = 30.000 deg,	R = 179.371 deg
};
P[176]{
   GP1:
	UF : 0, UT : 1,		CONFIG : 'N U T, 0, 0, 0',
	X = 1122.268  mm,	Y = -69.187  mm,	Z = -245.376  mm,
	W = 0.000 deg,	P = 30.000 deg,	R = 179.371 deg
};
P[177]{
   GP1:
	UF : 0, UT : 1,		CONFIG : 'N U T, 0, 0, 0',
	X = 1120.839  mm,	Y = -66.837  mm,	Z = -245.166  mm,
	W = 0.000 deg,	P = 30.000 deg,	R = 179.371 deg
};
P[178]{
   GP1:
	UF : 0, UT : 1,		CONFIG : 'N U T, 0, 0, 0',
	X = 1120.113  mm,	Y = -64.561  mm,	Z = -245.051  mm,
	W = 0.000 deg,	P = 30.000 deg,	R = 179.371 deg
};
P[179]{
   GP1:
	UF : 0, UT : 1,		CONFIG : 'N U T, 0, 0, 0',
	X = 1119.526  mm,	Y = -62.394  mm,	Z = -244.968  mm,
	W = 0.000 deg,	P = 30.000 deg,	R = 179.371 deg
};
P[180]{
   GP1:
	UF : 0, UT : 1,		CONFIG : 'N U T, 0, 0, 0',
	X = 1119.241  mm,	Y = -60.218  mm,	Z = -244.941  mm,
	W = 0.000 deg,	P = 30.000 deg,	R = 179.371 deg
};
P[181]{
   GP1:
	UF : 0, UT : 1,		CONFIG : 'N U T, 0, 0, 0',
	X = 1119.052  mm,	Y = -58.125  mm,	Z = -244.914  mm,
	W = 0.000 deg,	P = 30.000 deg,	R = 179.371 deg
};
P[182]{
   GP1:
	UF : 0, UT : 1,		CONFIG : 'N U T, 0, 0, 0',
	X = 1118.980  mm,	Y = -56.057  mm,	Z = -244.898  mm,
	W = 0.000 deg,	P = 30.000 deg,	R = 179.371 deg
};
P[183]{
   GP1:
	UF : 0, UT : 1,		CONFIG : 'N U T, 0, 0, 0',
	X = 1118.934  mm,	Y = -54.034  mm,	Z = -244.884  mm,
	W = 0.000 deg,	P = 30.000 deg,	R = 179.371 deg
};
P[184]{
   GP1:
	UF : 0, UT : 1,		CONFIG : 'N U T, 0, 0, 0',
	X = 1118.911  mm,	Y = -52.014  mm,	Z = -244.873  mm,
	W = 0.000 deg,	P = 30.000 deg,	R = 179.371 deg
};
P[185]{
   GP1:
	UF : 0, UT : 1,		CONFIG : 'N U T, 0, 0, 0',
	X = 1118.905  mm,	Y = -50.003  mm,	Z = -244.864  mm,
	W = 0.000 deg,	P = 30.000 deg,	R = 179.371 deg
};
P[186]{
   GP1:
	UF : 0, UT : 1,		CONFIG : 'N U T, 0, 0, 0',
	X = 1118.905  mm,	Y = -47.998  mm,	Z = -244.852  mm,
	W = 0.000 deg,	P = 30.000 deg,	R = 179.371 deg
};
P[187]{
   GP1:
	UF : 0, UT : 1,		CONFIG : 'N U T, 0, 0, 0',
	X = 1118.909  mm,	Y = -45.995  mm,	Z = -244.837  mm,
	W = 0.000 deg,	P = 30.000 deg,	R = 179.371 deg
};
P[188]{
   GP1:
	UF : 0, UT : 1,		CONFIG : 'N U T, 0, 0, 0',
	X = 1118.916  mm,	Y = -43.989  mm,	Z = -244.827  mm,
	W = 0.000 deg,	P = 30.000 deg,	R = 179.371 deg
};
P[189]{
   GP1:
	UF : 0, UT : 1,		CONFIG : 'N U T, 0, 0, 0',
	X = 1118.931  mm,	Y = -41.983  mm,	Z = -244.818  mm,
	W = 0.000 deg,	P = 30.000 deg,	R = 179.371 deg
};
P[190]{
   GP1:
	UF : 0, UT : 1,		CONFIG : 'N U T, 0, 0, 0',
	X = 1118.950  mm,	Y = -39.981  mm,	Z = -244.804  mm,
	W = 0.000 deg,	P = 30.000 deg,	R = 179.371 deg
};
P[191]{
   GP1:
	UF : 0, UT : 1,		CONFIG : 'N U T, 0, 0, 0',
	X = 1118.969  mm,	Y = -37.978  mm,	Z = -244.790  mm,
	W = 0.000 deg,	P = 30.000 deg,	R = 179.371 deg
};
P[192]{
   GP1:
	UF : 0, UT : 1,		CONFIG : 'N U T, 0, 0, 0',
	X = 1122.992  mm,	Y = -36.032  mm,	Z = -244.774  mm,
	W = 0.000 deg,	P = 30.000 deg,	R = 179.371 deg
};
P[193]{
   GP1:
	UF : 0, UT : 1,		CONFIG : 'N U T, 0, 0, 0',
	X = 1123.033  mm,	Y = -34.045  mm,	Z = -244.755  mm,
	W = 0.000 deg,	P = 30.000 deg,	R = 179.371 deg
};
P[194]{
   GP1:
	UF : 0, UT : 1,		CONFIG : 'N U T, 0, 0, 0',
	X = 1123.081  mm,	Y = -32.056  mm,	Z = -244.734  mm,
	W = 0.000 deg,	P = 30.000 deg,	R = 179.371 deg
};
P[195]{
   GP1:
	UF : 0, UT : 1,		CONFIG : 'N U T, 0, 0, 0',
	X = 1123.145  mm,	Y = -30.064  mm,	Z = -244.711  mm,
	W = 0.000 deg,	P = 30.000 deg,	R = 179.371 deg
};
P[196]{
   GP1:
	UF : 0, UT : 1,		CONFIG : 'N U T, 0, 0, 0',
	X = 1123.209  mm,	Y = -28.070  mm,	Z = -244.689  mm,
	W = 0.000 deg,	P = 30.000 deg,	R = 179.371 deg
};
P[197]{
   GP1:
	UF : 0, UT : 1,		CONFIG : 'N U T, 0, 0, 0',
	X = 1123.283  mm,	Y = -26.080  mm,	Z = -244.673  mm,
	W = 0.000 deg,	P = 30.000 deg,	R = 179.371 deg
};
P[198]{
   GP1:
	UF : 0, UT : 1,		CONFIG : 'N U T, 0, 0, 0',
	X = 1123.368  mm,	Y = -24.092  mm,	Z = -244.662  mm,
	W = 0.000 deg,	P = 30.000 deg,	R = 179.371 deg
};
P[199]{
   GP1:
	UF : 0, UT : 1,		CONFIG : 'N U T, 0, 0, 0',
	X = 1123.466  mm,	Y = -22.105  mm,	Z = -244.648  mm,
	W = 0.000 deg,	P = 30.000 deg,	R = 179.371 deg
};
P[200]{
   GP1:
	UF : 0, UT : 1,		CONFIG : 'N U T, 0, 0, 0',
	X = 1123.576  mm,	Y = -20.131  mm,	Z = -244.635  mm,
	W = 0.000 deg,	P = 30.000 deg,	R = 179.371 deg
};
P[201]{
   GP1:
	UF : 0, UT : 1,		CONFIG : 'N U T, 0, 0, 0',
	X = 1123.726  mm,	Y = -18.164  mm,	Z = -244.626  mm,
	W = 0.000 deg,	P = 30.000 deg,	R = 179.371 deg
};
P[202]{
   GP1:
	UF : 0, UT : 1,		CONFIG : 'N U T, 0, 0, 0',
	X = 1119.920  mm,	Y = -15.784  mm,	Z = -244.626  mm,
	W = 0.000 deg,	P = 30.000 deg,	R = 171.849 deg
};
P[203]{
   GP1:
	UF : 0, UT : 1,		CONFIG : 'N U T, 0, 0, 0',
	X = 1120.195  mm,	Y = -13.666  mm,	Z = -244.634  mm,
	W = 0.000 deg,	P = 30.000 deg,	R = 163.304 deg
};
P[204]{
   GP1:
	UF : 0, UT : 1,		CONFIG : 'N U T, 0, 0, 0',
	X = 1120.639  mm,	Y = -11.547  mm,	Z = -244.657  mm,
	W = 0.000 deg,	P = 30.000 deg,	R = 154.645 deg
};
P[205]{
   GP1:
	UF : 0, UT : 1,		CONFIG : 'N U T, 0, 0, 0',
	X = 1121.175  mm,	Y = -9.450  mm,	Z = -244.698  mm,
	W = 0.000 deg,	P = 30.000 deg,	R = 145.897 deg
};
P[206]{
   GP1:
	UF : 0, UT : 1,		CONFIG : 'N U T, 0, 0, 0',
	X = 1121.853  mm,	Y = -7.314  mm,	Z = -244.784  mm,
	W = 0.000 deg,	P = 30.000 deg,	R = 137.000 deg
};
P[207]{
   GP1:
	UF : 0, UT : 1,		CONFIG : 'N U T, 0, 0, 0',
	X = 1122.744  mm,	Y = -5.157  mm,	Z = -244.921  mm,
	W = 0.000 deg,	P = 30.000 deg,	R = 137.000 deg
};
P[208]{
   GP1:
	UF : 0, UT : 1,		CONFIG : 'N U T, 0, 0, 0',
	X = 1123.857  mm,	Y = -3.001  mm,	Z = -245.101  mm,
	W = 0.000 deg,	P = 30.000 deg,	R = 137.000 deg
};
P[209]{
   GP1:
	UF : 0, UT : 1,		CONFIG : 'N U T, 0, 0, 0',
	X = 1125.210  mm,	Y = -0.876  mm,	Z = -245.319  mm,
	W = 0.000 deg,	P = 30.000 deg,	R = 137.000 deg
};
P[210]{
   GP1:
	UF : 0, UT : 1,		CONFIG : 'N U T, 0, 0, 0',
	X = 1126.712  mm,	Y = 1.206  mm,	Z = -245.619  mm,
	W = 0.000 deg,	P = 30.000 deg,	R = 137.000 deg
};
P[211]{
   GP1:
	UF : 0, UT : 1,		CONFIG : 'N U T, 0, 0, 0',
	X = 1128.368  mm,	Y = 3.300  mm,	Z = -246.007  mm,
	W = 0.000 deg,	P = 30.000 deg,	R = 137.000 deg
};
P[212]{
   GP1:
	UF : 0, UT : 1,		CONFIG : 'N U T, 0, 0, 0',
	X = 1133.183  mm,	Y = 2.625  mm,	Z = -246.506  mm,
	W = 0.000 deg,	P = 30.000 deg,	R = 137.000 deg
};
P[213]{
   GP1:
	UF : 0, UT : 1,		CONFIG : 'N U T, 0, 0, 0',
	X = 1135.104  mm,	Y = 4.603  mm,	Z = -247.048  mm,
	W = 0.000 deg,	P = 30.000 deg,	R = 137.000 deg
};
P[214]{
   GP1:
	UF : 0, UT : 1,		CONFIG : 'N U T, 0, 0, 0',
	X = 1137.036  mm,	Y = 6.572  mm,	Z = -247.607  mm,
	W = 0.000 deg,	P = 30.000 deg,	R = 137.000 deg
};
P[215]{
   GP1:
	UF : 0, UT : 1,		CONFIG : 'N U T, 0, 0, 0',
	X = 1139.118  mm,	Y = 8.539  mm,	Z = -248.254  mm,
	W = 0.000 deg,	P = 30.000 deg,	R = 137.000 deg
};
P[216]{
   GP1:
	UF : 0, UT : 1,		CONFIG : 'N U T, 0, 0, 0',
	X = 1141.272  mm,	Y = 10.531  mm,	Z = -248.968  mm,
	W = 0.000 deg,	P = 30.000 deg,	R = 137.000 deg
};
P[217]{
   GP1:
	UF : 0, UT : 1,		CONFIG : 'N U T, 0, 0, 0',
	X = 1143.442  mm,	Y = 12.534  mm,	Z = -249.668  mm,
	W = 0.000 deg,	P = 30.000 deg,	R = 137.000 deg
};
P[218]{
   GP1:
	UF : 0, UT : 1,		CONFIG : 'N U T, 0, 0, 0',
	X = 1145.599  mm,	Y = 14.548  mm,	Z = -250.350  mm,
	W = 0.000 deg,	P = 30.000 deg,	R = 140.970 deg
};
P[219]{
   GP1:
	UF : 0, UT : 1,		CONFIG : 'N U T, 0, 0, 0',
	X = 1147.678  mm,	Y = 16.544  mm,	Z = -250.985  mm,
	W = 0.000 deg,	P = 30.000 deg,	R = 152.690 deg
};
P[220]{
   GP1:
	UF : 0, UT : 1,		CONFIG : 'N U T, 0, 0, 0',
	X = 1149.827  mm,	Y = 18.530  mm,	Z = -251.634  mm,
	W = 0.000 deg,	P = 30.000 deg,	R = 164.650 deg
};
P[221]{
   GP1:
	UF : 0, UT : 1,		CONFIG : 'N U T, 0, 0, 0',
	X = 1152.045  mm,	Y = 20.575  mm,	Z = -252.294  mm,
	W = 0.000 deg,	P = 30.000 deg,	R = 176.637 deg
};
P[222]{
   GP1:
	UF : 0, UT : 1,		CONFIG : 'N U T, 0, 0, 0',
	X = 1154.021  mm,	Y = 22.663  mm,	Z = -252.858  mm,
	W = 0.000 deg,	P = 30.000 deg,	R = 176.637 deg
};
P[223]{
   GP1:
	UF : 0, UT : 1,		CONFIG : 'N U T, 0, 0, 0',
	X = 1155.800  mm,	Y = 24.754  mm,	Z = -253.352  mm,
	W = 0.000 deg,	P = 30.000 deg,	R = 176.637 deg
};
P[224]{
   GP1:
	UF : 0, UT : 1,		CONFIG : 'N U T, 0, 0, 0',
	X = 1157.378  mm,	Y = 26.881  mm,	Z = -253.775  mm,
	W = 0.000 deg,	P = 30.000 deg,	R = 176.637 deg
};
P[225]{
   GP1:
	UF : 0, UT : 1,		CONFIG : 'N U T, 0, 0, 0',
	X = 1158.702  mm,	Y = 29.060  mm,	Z = -254.115  mm,
	W = 0.000 deg,	P = 30.000 deg,	R = 176.637 deg
};
P[226]{
   GP1:
	UF : 0, UT : 1,		CONFIG : 'N U T, 0, 0, 0',
	X = 1159.722  mm,	Y = 31.292  mm,	Z = -254.372  mm,
	W = 0.000 deg,	P = 30.000 deg,	R = 176.637 deg
};
P[227]{
   GP1:
	UF : 0, UT : 1,		CONFIG : 'N U T, 0, 0, 0',
	X = 1160.397  mm,	Y = 33.537  mm,	Z = -254.534  mm,
	W = 0.000 deg,	P = 30.000 deg,	R = 176.637 deg
};
P[228]{
   GP1:
	UF : 0, UT : 1,		CONFIG : 'N U T, 0, 0, 0',
	X = 1160.782  mm,	Y = 35.715  mm,	Z = -254.620  mm,
	W = 0.000 deg,	P = 30.000 deg,	R = 176.637 deg
};
P[229]{
   GP1:
	UF : 0, UT : 1,		CONFIG : 'N U T, 0, 0, 0',
	X = 1161.021  mm,	Y = 37.841  mm,	Z = -254.669  mm,
	W = 0.000 deg,	P = 30.000 deg,	R = 176.637 deg
};
P[230]{
   GP1:
	UF : 0, UT : 1,		CONFIG : 'N U T, 0, 0, 0',
	X = 1157.123  mm,	Y = 40.074  mm,	Z = -254.678  mm,
	W = 0.000 deg,	P = 30.000 deg,	R = 176.637 deg
};
P[231]{
   GP1:
	UF : 0, UT : 1,		CONFIG : 'N U T, 0, 0, 0',
	X = 1157.175  mm,	Y = 42.045  mm,	Z = -254.676  mm,
	W = 0.000 deg,	P = 30.000 deg,	R = 176.637 deg
};
P[232]{
   GP1:
	UF : 0, UT : 1,		CONFIG : 'N U T, 0, 0, 0',
	X = 1157.212  mm,	Y = 44.034  mm,	Z = -254.671  mm,
	W = 0.000 deg,	P = 30.000 deg,	R = 176.637 deg
};
P[233]{
   GP1:
	UF : 0, UT : 1,		CONFIG : 'N U T, 0, 0, 0',
	X = 1157.243  mm,	Y = 46.028  mm,	Z = -254.658  mm,
	W = 0.000 deg,	P = 30.000 deg,	R = 176.637 deg
};
P[234]{
   GP1:
	UF : 0, UT : 1,		CONFIG : 'N U T, 0, 0, 0',
	X = 1157.268  mm,	Y = 48.024  mm,	Z = -254.640  mm,
	W = 0.000 deg,	P = 30.000 deg,	R = 176.637 deg
};
P[235]{
   GP1:
	UF : 0, UT : 1,		CONFIG : 'N U T, 0, 0, 0',
	X = 1157.291  mm,	Y = 50.020  mm,	Z = -254.621  mm,
	W = 0.000 deg,	P = 30.000 deg,	R = 176.637 deg
};
P[236]{
   GP1:
	UF : 0, UT : 1,		CONFIG : 'N U T, 0, 0, 0',
	X = 1157.307  mm,	Y = 52.011  mm,	Z = -254.598  mm,
	W = 0.000 deg,	P = 30.000 deg,	R = 176.637 deg
};
P[237]{
   GP1:
	UF : 0, UT : 1,		CONFIG : 'N U T, 0, 0, 0',
	X = 1157.313  mm,	Y = 54.001  mm,	Z = -254.575  mm,
	W = 0.000 deg,	P = 30.000 deg,	R = 176.637 deg
};
P[238]{
   GP1:
	UF : 0, UT : 1,		CONFIG : 'N U T, 0, 0, 0',
	X = 1157.310  mm,	Y = 55.994  mm,	Z = -254.550  mm,
	W = 0.000 deg,	P = 30.000 deg,	R = 176.637 deg
};
P[239]{
   GP1:
	UF : 0, UT : 1,		CONFIG : 'N U T, 0, 0, 0',
	X = 1157.301  mm,	Y = 57.988  mm,	Z = -254.518  mm,
	W = 0.000 deg,	P = 30.000 deg,	R = 176.637 deg
};
P[240]{
   GP1:
	UF : 0, UT : 1,		CONFIG : 'N U T, 0, 0, 0',
	X = 1157.286  mm,	Y = 59.983  mm,	Z = -254.491  mm,
	W = 0.000 deg,	P = 30.000 deg,	R = 176.637 deg
};
P[241]{
   GP1:
	UF : 0, UT : 1,		CONFIG : 'N U T, 0, 0, 0',
	X = 1157.267  mm,	Y = 61.975  mm,	Z = -254.460  mm,
	W = 0.000 deg,	P = 30.000 deg,	R = 176.637 deg
};
P[242]{
   GP1:
	UF : 0, UT : 1,		CONFIG : 'N U T, 0, 0, 0',
	X = 1157.237  mm,	Y = 63.966  mm,	Z = -254.428  mm,
	W = 0.000 deg,	P = 30.000 deg,	R = 176.637 deg
};
P[243]{
   GP1:
	UF : 0, UT : 1,		CONFIG : 'N U T, 0, 0, 0',
	X = 1157.200  mm,	Y = 65.957  mm,	Z = -254.394  mm,
	W = 0.000 deg,	P = 30.000 deg,	R = 176.637 deg
};
P[244]{
   GP1:
	UF : 0, UT : 1,		CONFIG : 'N U T, 0, 0, 0',
	X = 1157.152  mm,	Y = 67.948  mm,	Z = -254.356  mm,
	W = 0.000 deg,	P = 30.000 deg,	R = 176.637 deg
};
P[245]{
   GP1:
	UF : 0, UT : 1,		CONFIG : 'N U T, 0, 0, 0',
	X = 1157.097  mm,	Y = 69.941  mm,	Z = -254.322  mm,
	W = 0.000 deg,	P = 30.000 deg,	R = 176.637 deg
};
P[246]{
   GP1:
	UF : 0, UT : 1,		CONFIG : 'N U T, 0, 0, 0',
	X = 1157.035  mm,	Y = 71.933  mm,	Z = -254.287  mm,
	W = 0.000 deg,	P = 30.000 deg,	R = 176.637 deg
};
P[247]{
   GP1:
	UF : 0, UT : 1,		CONFIG : 'N U T, 0, 0, 0',
	X = 1156.964  mm,	Y = 73.923  mm,	Z = -254.246  mm,
	W = 0.000 deg,	P = 30.000 deg,	R = 176.637 deg
};
P[248]{
   GP1:
	UF : 0, UT : 1,		CONFIG : 'N U T, 0, 0, 0',
	X = 1156.882  mm,	Y = 75.915  mm,	Z = -254.204  mm,
	W = 0.000 deg,	P = 30.000 deg,	R = 176.637 deg
};
P[249]{
   GP1:
	UF : 0, UT : 1,		CONFIG : 'N U T, 0, 0, 0',
	X = 1156.794  mm,	Y = 77.905  mm,	Z = -254.160  mm,
	W = 0.000 deg,	P = 30.000 deg,	R = 176.637 deg
};
P[250]{
   GP1:
	UF : 0, UT : 1,		CONFIG : 'N U T, 0, 0, 0',
	X = 1160.686  mm,	Y = 80.124  mm,	Z = -254.112  mm,
	W = 0.000 deg,	P = 30.000 deg,	R = -174.658 deg
};
P[251]{
   GP1:
	UF : 0, UT : 1,		CONFIG : 'N U T, 0, 0, 0',
	X = 1160.535  mm,	Y = 82.172  mm,	Z = -254.053  mm,
	W = 0.000 deg,	P = 30.000 deg,	R = -165.137 deg
};
P[252]{
   GP1:
	UF : 0, UT : 1,		CONFIG : 'N U T, 0, 0, 0',
	X = 1160.318  mm,	Y = 84.323  mm,	Z = -253.973  mm,
	W = 0.000 deg,	P = 30.000 deg,	R = -155.591 deg
};
P[253]{
   GP1:
	UF : 0, UT : 1,		CONFIG : 'N U T, 0, 0, 0',
	X = 1159.825  mm,	Y = 86.500  mm,	Z = -253.817  mm,
	W = 0.000 deg,	P = 30.000 deg,	R = -145.829 deg
};
P[254]{
   GP1:
	UF : 0, UT : 1,		CONFIG : 'N U T, 0, 0, 0',
	X = 1159.187  mm,	Y = 88.693  mm,	Z = -253.622  mm,
	W = 0.000 deg,	P = 30.000 deg,	R = -135.906 deg
};
P[255]{
   GP1:
	UF : 0, UT : 1,		CONFIG : 'N U T, 0, 0, 0',
	X = 1158.199  mm,	Y = 90.898  mm,	Z = -253.324  mm,
	W = 0.000 deg,	P = 30.000 deg,	R = -135.906 deg
};
P[256]{
   GP1:
	UF : 0, UT : 1,		CONFIG : 'N U T, 0, 0, 0',
	X = 1156.991  mm,	Y = 93.072  mm,	Z = -252.965  mm,
	W = 0.000 deg,	P = 30.000 deg,	R = -135.906 deg
};
P[257]{
   GP1:
	UF : 0, UT : 1,		CONFIG : 'N U T, 0, 0, 0',
	X = 1155.439  mm,	Y = 95.244  mm,	Z = -252.507  mm,
	W = 0.000 deg,	P = 30.000 deg,	R = -135.906 deg
};
P[258]{
   GP1:
	UF : 0, UT : 1,		CONFIG : 'N U T, 0, 0, 0',
	X = 1150.704  mm,	Y = 94.594  mm,	Z = -251.931  mm,
	W = 0.000 deg,	P = 30.000 deg,	R = -135.906 deg
};
P[259]{
   GP1:
	UF : 0, UT : 1,		CONFIG : 'N U T, 0, 0, 0',
	X = 1148.558  mm,	Y = 96.533  mm,	Z = -251.204  mm,
	W = 0.000 deg,	P = 30.000 deg,	R = -135.906 deg
};
P[260]{
   GP1:
	UF : 0, UT : 1,		CONFIG : 'N U T, 0, 0, 0',
	X = 1146.452  mm,	Y = 98.531  mm,	Z = -250.510  mm,
	W = 0.000 deg,	P = 30.000 deg,	R = -135.906 deg
};
P[261]{
   GP1:
	UF : 0, UT : 1,		CONFIG : 'N U T, 0, 0, 0',
	X = 1144.202  mm,	Y = 100.561  mm,	Z = -249.773  mm,
	W = 0.000 deg,	P = 30.000 deg,	R = -135.906 deg
};
P[262]{
   GP1:
	UF : 0, UT : 1,		CONFIG : 'N U T, 0, 0, 0',
	X = 1142.252  mm,	Y = 102.586  mm,	Z = -249.132  mm,
	W = 0.000 deg,	P = 30.000 deg,	R = -135.906 deg
};
P[263]{
   GP1:
	UF : 0, UT : 1,		CONFIG : 'N U T, 0, 0, 0',
	X = 1140.229  mm,	Y = 104.536  mm,	Z = -248.421  mm,
	W = 0.000 deg,	P = 30.000 deg,	R = -135.906 deg
};
P[264]{
   GP1:
	UF : 0, UT : 1,		CONFIG : 'N U T, 0, 0, 0',
	X = 1138.009  mm,	Y = 106.536  mm,	Z = -247.684  mm,
	W = 0.000 deg,	P = 30.000 deg,	R = -135.906 deg
};
P[265]{
   GP1:
	UF : 0, UT : 1,		CONFIG : 'N U T, 0, 0, 0',
	X = 1135.980  mm,	Y = 108.491  mm,	Z = -246.991  mm,
	W = 0.000 deg,	P = 30.000 deg,	R = -135.906 deg
};
P[266]{
   GP1:
	UF : 0, UT : 1,		CONFIG : 'N U T, 0, 0, 0',
	X = 1133.514  mm,	Y = 110.447  mm,	Z = -246.351  mm,
	W = 0.000 deg,	P = 30.000 deg,	R = -135.906 deg
};
P[267]{
   GP1:
	UF : 0, UT : 1,		CONFIG : 'N U T, 0, 0, 0',
	X = 1131.049  mm,	Y = 112.490  mm,	Z = -245.753  mm,
	W = 0.000 deg,	P = 30.000 deg,	R = -135.906 deg
};
P[268]{
   GP1:
	UF : 0, UT : 1,		CONFIG : 'N U T, 0, 0, 0',
	X = 1128.830  mm,	Y = 114.517  mm,	Z = -245.193  mm,
	W = 0.000 deg,	P = 30.000 deg,	R = -143.887 deg
};
P[269]{
   GP1:
	UF : 0, UT : 1,		CONFIG : 'N U T, 0, 0, 0',
	X = 1126.545  mm,	Y = 116.567  mm,	Z = -244.621  mm,
	W = 0.000 deg,	P = 30.000 deg,	R = -158.130 deg
};
P[270]{
   GP1:
	UF : 0, UT : 1,		CONFIG : 'N U T, 0, 0, 0',
	X = 1124.519  mm,	Y = 118.732  mm,	Z = -244.178  mm,
	W = 0.000 deg,	P = 30.000 deg,	R = -171.094 deg
};
P[271]{
   GP1:
	UF : 0, UT : 1,		CONFIG : 'N U T, 0, 0, 0',
	X = 1122.985  mm,	Y = 120.911  mm,	Z = -243.864  mm,
	W = 0.000 deg,	P = 30.000 deg,	R = 177.406 deg
};
P[272]{
   GP1:
	UF : 0, UT : 1,		CONFIG : 'N U T, 0, 0, 0',
	X = 1121.587  mm,	Y = 123.328  mm,	Z = -243.635  mm,
	W = 0.000 deg,	P = 30.000 deg,	R = 177.406 deg
};
P[273]{
   GP1:
	UF : 0, UT : 1,		CONFIG : 'N U T, 0, 0, 0',
	X = 1121.246  mm,	Y = 125.794  mm,	Z = -243.520  mm,
	W = 0.000 deg,	P = 30.000 deg,	R = 177.406 deg
};
P[274]{
   GP1:
	UF : 0, UT : 1,		CONFIG : 'N U T, 0, 0, 0',
	X = 1121.064  mm,	Y = 127.833  mm,	Z = -243.408  mm,
	W = 0.000 deg,	P = 30.000 deg,	R = 177.406 deg
};
P[275]{
   GP1:
	UF : 0, UT : 1,		CONFIG : 'N U T, 0, 0, 0',
	X = 1120.904  mm,	Y = 129.884  mm,	Z = -243.348  mm,
	W = 0.000 deg,	P = 30.000 deg,	R = 177.406 deg
};
P[276]{
   GP1:
	UF : 0, UT : 1,		CONFIG : 'N U T, 0, 0, 0',
	X = 1120.827  mm,	Y = 131.933  mm,	Z = -243.310  mm,
	W = 0.000 deg,	P = 30.000 deg,	R = 177.406 deg
};
P[277]{
   GP1:
	UF : 0, UT : 1,		CONFIG : 'N U T, 0, 0, 0',
	X = 1120.768  mm,	Y = 133.949  mm,	Z = -243.270  mm,
	W = 0.000 deg,	P = 30.000 deg,	R = 177.406 deg
};
P[278]{
   GP1:
	UF : 0, UT : 1,		CONFIG : 'N U T, 0, 0, 0',
	X = 1120.724  mm,	Y = 135.965  mm,	Z = -243.231  mm,
	W = 0.000 deg,	P = 30.000 deg,	R = 177.406 deg
};
P[279]{
   GP1:
	UF : 0, UT : 1,		CONFIG : 'N U T, 0, 0, 0',
	X = 1120.697  mm,	Y = 137.978  mm,	Z = -243.199  mm,
	W = 0.000 deg,	P = 30.000 deg,	R = 177.406 deg
};
P[280]{
   GP1:
	UF : 0, UT : 1,		CONFIG : 'N U T, 0, 0, 0',
	X = 1120.679  mm,	Y = 139.988  mm,	Z = -243.170  mm,
	W = 0.000 deg,	P = 30.000 deg,	R = 177.406 deg
};
P[281]{
   GP1:
	UF : 0, UT : 1,		CONFIG : 'N U T, 0, 0, 0',
	X = 1120.673  mm,	Y = 141.995  mm,	Z = -243.128  mm,
	W = 0.000 deg,	P = 30.000 deg,	R = 177.406 deg
};
P[282]{
   GP1:
	UF : 0, UT : 1,		CONFIG : 'N U T, 0, 0, 0',
	X = 1120.669  mm,	Y = 143.999  mm,	Z = -243.084  mm,
	W = 0.000 deg,	P = 30.000 deg,	R = 177.406 deg
};
P[283]{
   GP1:
	UF : 0, UT : 1,		CONFIG : 'N U T, 0, 0, 0',
	X = 1120.671  mm,	Y = 146.015  mm,	Z = -243.043  mm,
	W = 0.000 deg,	P = 30.000 deg,	R = 177.406 deg
};
P[284]{
   GP1:
	UF : 0, UT : 1,		CONFIG : 'N U T, 0, 0, 0',
	X = 1120.698  mm,	Y = 148.032  mm,	Z = -243.008  mm,
	W = 0.000 deg,	P = 30.000 deg,	R = 177.406 deg
};
P[285]{
   GP1:
	UF : 0, UT : 1,		CONFIG : 'N U T, 0, 0, 0',
	X = 1120.736  mm,	Y = 150.043  mm,	Z = -242.976  mm,
	W = 0.000 deg,	P = 30.000 deg,	R = 177.406 deg
};
P[286]{
   GP1:
	UF : 0, UT : 1,		CONFIG : 'N U T, 0, 0, 0',
	X = 1120.784  mm,	Y = 152.048  mm,	Z = -242.943  mm,
	W = 0.000 deg,	P = 30.000 deg,	R = 177.406 deg
};
P[287]{
   GP1:
	UF : 0, UT : 1,		CONFIG : 'N U T, 0, 0, 0',
	X = 1120.833  mm,	Y = 154.057  mm,	Z = -242.915  mm,
	W = 0.000 deg,	P = 30.000 deg,	R = 177.406 deg
};
P[288]{
   GP1:
	UF : 0, UT : 1,		CONFIG : 'N U T, 0, 0, 0',
	X = 1120.899  mm,	Y = 156.067  mm,	Z = -242.907  mm,
	W = 0.000 deg,	P = 30.000 deg,	R = 177.406 deg
};
P[289]{
   GP1:
	UF : 0, UT : 1,		CONFIG : 'N U T, 0, 0, 0',
	X = 1120.968  mm,	Y = 158.076  mm,	Z = -242.901  mm,
	W = 0.000 deg,	P = 30.000 deg,	R = 177.406 deg
};
P[290]{
   GP1:
	UF : 0, UT : 1,		CONFIG : 'N U T, 0, 0, 0',
	X = 1121.052  mm,	Y = 160.080  mm,	Z = -242.900  mm,
	W = 0.000 deg,	P = 30.000 deg,	R = 177.406 deg
};
P[291]{
   GP1:
	UF : 0, UT : 1,		CONFIG : 'N U T, 0, 0, 0',
	X = 1121.128  mm,	Y = 162.088  mm,	Z = -242.905  mm,
	W = 0.000 deg,	P = 30.000 deg,	R = 177.406 deg
};
P[292]{
   GP1:
	UF : 0, UT : 1,		CONFIG : 'N U T, 0, 0, 0',
	X = 1125.224  mm,	Y = 163.900  mm,	Z = -242.916  mm,
	W = 0.000 deg,	P = 30.000 deg,	R = 177.406 deg
};
P[293]{
   GP1:
	UF : 0, UT : 1,		CONFIG : 'N U T, 0, 0, 0',
	X = 1125.323  mm,	Y = 165.878  mm,	Z = -242.928  mm,
	W = 0.000 deg,	P = 30.000 deg,	R = 177.406 deg
};
P[294]{
   GP1:
	UF : 0, UT : 1,		CONFIG : 'N U T, 0, 0, 0',
	X = 1125.466  mm,	Y = 167.850  mm,	Z = -242.939  mm,
	W = 0.000 deg,	P = 30.000 deg,	R = 177.406 deg
};
P[295]{
   GP1:
	UF : 0, UT : 1,		CONFIG : 'N U T, 0, 0, 0',
	X = 1125.619  mm,	Y = 169.821  mm,	Z = -242.949  mm,
	W = 0.000 deg,	P = 30.000 deg,	R = 177.406 deg
};
P[296]{
   GP1:
	UF : 0, UT : 1,		CONFIG : 'N U T, 0, 0, 0',
	X = 1121.841  mm,	Y = 172.204  mm,	Z = -242.963  mm,
	W = 0.000 deg,	P = 30.000 deg,	R = 170.014 deg
};
P[297]{
   GP1:
	UF : 0, UT : 1,		CONFIG : 'N U T, 0, 0, 0',
	X = 1122.053  mm,	Y = 174.244  mm,	Z = -242.981  mm,
	W = 0.000 deg,	P = 30.000 deg,	R = 161.910 deg
};
P[298]{
   GP1:
	UF : 0, UT : 1,		CONFIG : 'N U T, 0, 0, 0',
	X = 1122.355  mm,	Y = 176.360  mm,	Z = -242.997  mm,
	W = 0.000 deg,	P = 30.000 deg,	R = 153.768 deg
};
P[299]{
   GP1:
	UF : 0, UT : 1,		CONFIG : 'N U T, 0, 0, 0',
	X = 1122.833  mm,	Y = 178.502  mm,	Z = -243.018  mm,
	W = 0.000 deg,	P = 30.000 deg,	R = 145.508 deg
};
P[300]{
   GP1:
	UF : 0, UT : 1,		CONFIG : 'N U T, 0, 0, 0',
	X = 1123.461  mm,	Y = 180.631  mm,	Z = -243.067  mm,
	W = 0.000 deg,	P = 30.000 deg,	R = 137.102 deg
};
P[301]{
   GP1:
	UF : 0, UT : 1,		CONFIG : 'N U T, 0, 0, 0',
	X = 1124.258  mm,	Y = 182.783  mm,	Z = -243.164  mm,
	W = 0.000 deg,	P = 30.000 deg,	R = 137.102 deg
};
P[302]{
   GP1:
	UF : 0, UT : 1,		CONFIG : 'N U T, 0, 0, 0',
	X = 1125.301  mm,	Y = 184.951  mm,	Z = -243.340  mm,
	W = 0.000 deg,	P = 30.000 deg,	R = 137.102 deg
};
P[303]{
   GP1:
	UF : 0, UT : 1,		CONFIG : 'N U T, 0, 0, 0',
	X = 1126.591  mm,	Y = 187.102  mm,	Z = -243.578  mm,
	W = 0.000 deg,	P = 30.000 deg,	R = 137.102 deg
};
P[304]{
   GP1:
	UF : 0, UT : 1,		CONFIG : 'N U T, 0, 0, 0',
	X = 1128.112  mm,	Y = 189.214  mm,	Z = -243.849  mm,
	W = 0.000 deg,	P = 30.000 deg,	R = 137.102 deg
};
P[305]{
   GP1:
	UF : 0, UT : 1,		CONFIG : 'N U T, 0, 0, 0',
	X = 1129.792  mm,	Y = 191.295  mm,	Z = -244.187  mm,
	W = 0.000 deg,	P = 30.000 deg,	R = 137.102 deg
};
P[306]{
   GP1:
	UF : 0, UT : 1,		CONFIG : 'N U T, 0, 0, 0',
	X = 1131.631  mm,	Y = 193.358  mm,	Z = -244.645  mm,
	W = 0.000 deg,	P = 30.000 deg,	R = 137.102 deg
};
P[307]{
   GP1:
	UF : 0, UT : 1,		CONFIG : 'N U T, 0, 0, 0',
	X = 1136.429  mm,	Y = 192.584  mm,	Z = -245.179  mm,
	W = 0.000 deg,	P = 30.000 deg,	R = 137.102 deg
};
P[308]{
   GP1:
	UF : 0, UT : 1,		CONFIG : 'N U T, 0, 0, 0',
	X = 1138.497  mm,	Y = 194.561  mm,	Z = -245.789  mm,
	W = 0.000 deg,	P = 30.000 deg,	R = 137.102 deg
};
P[309]{
   GP1:
	UF : 0, UT : 1,		CONFIG : 'N U T, 0, 0, 0',
	X = 1140.547  mm,	Y = 196.557  mm,	Z = -246.387  mm,
	W = 0.000 deg,	P = 30.000 deg,	R = 137.102 deg
};
P[310]{
   GP1:
	UF : 0, UT : 1,		CONFIG : 'N U T, 0, 0, 0',
	X = 1142.623  mm,	Y = 198.522  mm,	Z = -247.028  mm,
	W = 0.000 deg,	P = 30.000 deg,	R = 137.102 deg
};
P[311]{
   GP1:
	UF : 0, UT : 1,		CONFIG : 'N U T, 0, 0, 0',
	X = 1144.885  mm,	Y = 200.510  mm,	Z = -247.765  mm,
	W = 0.000 deg,	P = 30.000 deg,	R = 140.074 deg
};
P[312]{
   GP1:
	UF : 0, UT : 1,		CONFIG : 'N U T, 0, 0, 0',
	X = 1147.099  mm,	Y = 202.530  mm,	Z = -248.488  mm,
	W = 0.000 deg,	P = 30.000 deg,	R = 150.242 deg
};
P[313]{
   GP1:
	UF : 0, UT : 1,		CONFIG : 'N U T, 0, 0, 0',
	X = 1149.246  mm,	Y = 204.531  mm,	Z = -249.179  mm,
	W = 0.000 deg,	P = 30.000 deg,	R = 160.273 deg
};
P[314]{
   GP1:
	UF : 0, UT : 1,		CONFIG : 'N U T, 0, 0, 0',
	X = 1151.447  mm,	Y = 206.547  mm,	Z = -249.866  mm,
	W = 0.000 deg,	P = 30.000 deg,	R = 170.392 deg
};
P[315]{
   GP1:
	UF : 0, UT : 1,		CONFIG : 'N U T, 0, 0, 0',
	X = 1153.496  mm,	Y = 208.552  mm,	Z = -250.497  mm,
	W = 0.000 deg,	P = 30.000 deg,	R = 170.392 deg
};
P[316]{
   GP1:
	UF : 0, UT : 1,		CONFIG : 'N U T, 0, 0, 0',
	X = 1155.674  mm,	Y = 210.577  mm,	Z = -251.159  mm,
	W = 0.000 deg,	P = 30.000 deg,	R = 170.392 deg
};
P[317]{
   GP1:
	UF : 0, UT : 1,		CONFIG : 'N U T, 0, 0, 0',
	X = 1157.680  mm,	Y = 212.692  mm,	Z = -251.747  mm,
	W = 0.000 deg,	P = 30.000 deg,	R = 170.392 deg
};
P[318]{
   GP1:
	UF : 0, UT : 1,		CONFIG : 'N U T, 0, 0, 0',
	X = 1159.333  mm,	Y = 214.809  mm,	Z = -252.210  mm,
	W = 0.000 deg,	P = 30.000 deg,	R = 170.392 deg
};
P[319]{
   GP1:
	UF : 0, UT : 1,		CONFIG : 'N U T, 0, 0, 0',
	X = 1160.827  mm,	Y = 216.941  mm,	Z = -252.617  mm,
	W = 0.000 deg,	P = 30.000 deg,	R = 170.392 deg
};
P[320]{
   GP1:
	UF : 0, UT : 1,		CONFIG : 'N U T, 0, 0, 0',
	X = 1162.036  mm,	Y = 219.155  mm,	Z = -252.930  mm,
	W = 0.000 deg,	P = 30.000 deg,	R = 170.392 deg
};
P[321]{
   GP1:
	UF : 0, UT : 1,		CONFIG : 'N U T, 0, 0, 0',
	X = 1162.894  mm,	Y = 221.377  mm,	Z = -253.146  mm,
	W = 0.000 deg,	P = 30.000 deg,	R = 170.392 deg
};
P[322]{
   GP1:
	UF : 0, UT : 1,		CONFIG : 'N U T, 0, 0, 0',
	X = 1163.499  mm,	Y = 223.630  mm,	Z = -253.290  mm,
	W = 0.000 deg,	P = 30.000 deg,	R = 170.392 deg
};
P[323]{
   GP1:
	UF : 0, UT : 1,		CONFIG : 'N U T, 0, 0, 0',
	X = 1159.753  mm,	Y = 226.164  mm,	Z = -253.336  mm,
	W = 0.000 deg,	P = 30.000 deg,	R = 170.392 deg
};
P[324]{
   GP1:
	UF : 0, UT : 1,		CONFIG : 'N U T, 0, 0, 0',
	X = 1159.864  mm,	Y = 228.069  mm,	Z = -253.340  mm,
	W = 0.000 deg,	P = 30.000 deg,	R = 170.392 deg
};
P[325]{
   GP1:
	UF : 0, UT : 1,		CONFIG : 'N U T, 0, 0, 0',
	X = 1159.885  mm,	Y = 230.004  mm,	Z = -253.333  mm,
	W = 0.000 deg,	P = 30.000 deg,	R = 170.392 deg
};
P[326]{
   GP1:
	UF : 0, UT : 1,		CONFIG : 'N U T, 0, 0, 0',
	X = 1159.870  mm,	Y = 231.982  mm,	Z = -253.323  mm,
	W = 0.000 deg,	P = 30.000 deg,	R = 170.392 deg
};
P[327]{
   GP1:
	UF : 0, UT : 1,		CONFIG : 'N U T, 0, 0, 0',
	X = 1159.849  mm,	Y = 233.979  mm,	Z = -253.310  mm,
	W = 0.000 deg,	P = 30.000 deg,	R = 170.392 deg
};
P[328]{
   GP1:
	UF : 0, UT : 1,		CONFIG : 'N U T, 0, 0, 0',
	X = 1159.827  mm,	Y = 235.976  mm,	Z = -253.290  mm,
	W = 0.000 deg,	P = 30.000 deg,	R = 170.392 deg
};
P[329]{
   GP1:
	UF : 0, UT : 1,		CONFIG : 'N U T, 0, 0, 0',
	X = 1159.802  mm,	Y = 237.971  mm,	Z = -253.263  mm,
	W = 0.000 deg,	P = 30.000 deg,	R = 170.392 deg
};
P[330]{
   GP1:
	UF : 0, UT : 1,		CONFIG : 'N U T, 0, 0, 0',
	X = 1159.770  mm,	Y = 239.967  mm,	Z = -253.226  mm,
	W = 0.000 deg,	P = 30.000 deg,	R = 170.392 deg
};
P[331]{
   GP1:
	UF : 0, UT : 1,		CONFIG : 'N U T, 0, 0, 0',
	X = 1159.736  mm,	Y = 241.967  mm,	Z = -253.186  mm,
	W = 0.000 deg,	P = 30.000 deg,	R = 170.392 deg
};
P[332]{
   GP1:
	UF : 0, UT : 1,		CONFIG : 'N U T, 0, 0, 0',
	X = 1159.704  mm,	Y = 243.969  mm,	Z = -253.149  mm,
	W = 0.000 deg,	P = 30.000 deg,	R = 170.392 deg
};
P[333]{
   GP1:
	UF : 0, UT : 1,		CONFIG : 'N U T, 0, 0, 0',
	X = 1159.673  mm,	Y = 245.968  mm,	Z = -253.110  mm,
	W = 0.000 deg,	P = 30.000 deg,	R = 170.392 deg
};
P[334]{
   GP1:
	UF : 0, UT : 1,		CONFIG : 'N U T, 0, 0, 0',
	X = 1159.641  mm,	Y = 247.959  mm,	Z = -253.068  mm,
	W = 0.000 deg,	P = 30.000 deg,	R = 170.392 deg
};
P[335]{
   GP1:
	UF : 0, UT : 1,		CONFIG : 'N U T, 0, 0, 0',
	X = 1159.592  mm,	Y = 249.952  mm,	Z = -253.021  mm,
	W = 0.000 deg,	P = 30.000 deg,	R = 170.392 deg
};
P[336]{
   GP1:
	UF : 0, UT : 1,		CONFIG : 'N U T, 0, 0, 0',
	X = 1159.545  mm,	Y = 251.953  mm,	Z = -252.981  mm,
	W = 0.000 deg,	P = 30.000 deg,	R = 170.392 deg
};
P[337]{
   GP1:
	UF : 0, UT : 1,		CONFIG : 'N U T, 0, 0, 0',
	X = 1159.499  mm,	Y = 253.954  mm,	Z = -252.951  mm,
	W = 0.000 deg,	P = 30.000 deg,	R = 170.392 deg
};
/END
